REGION Network 20: Panel 20
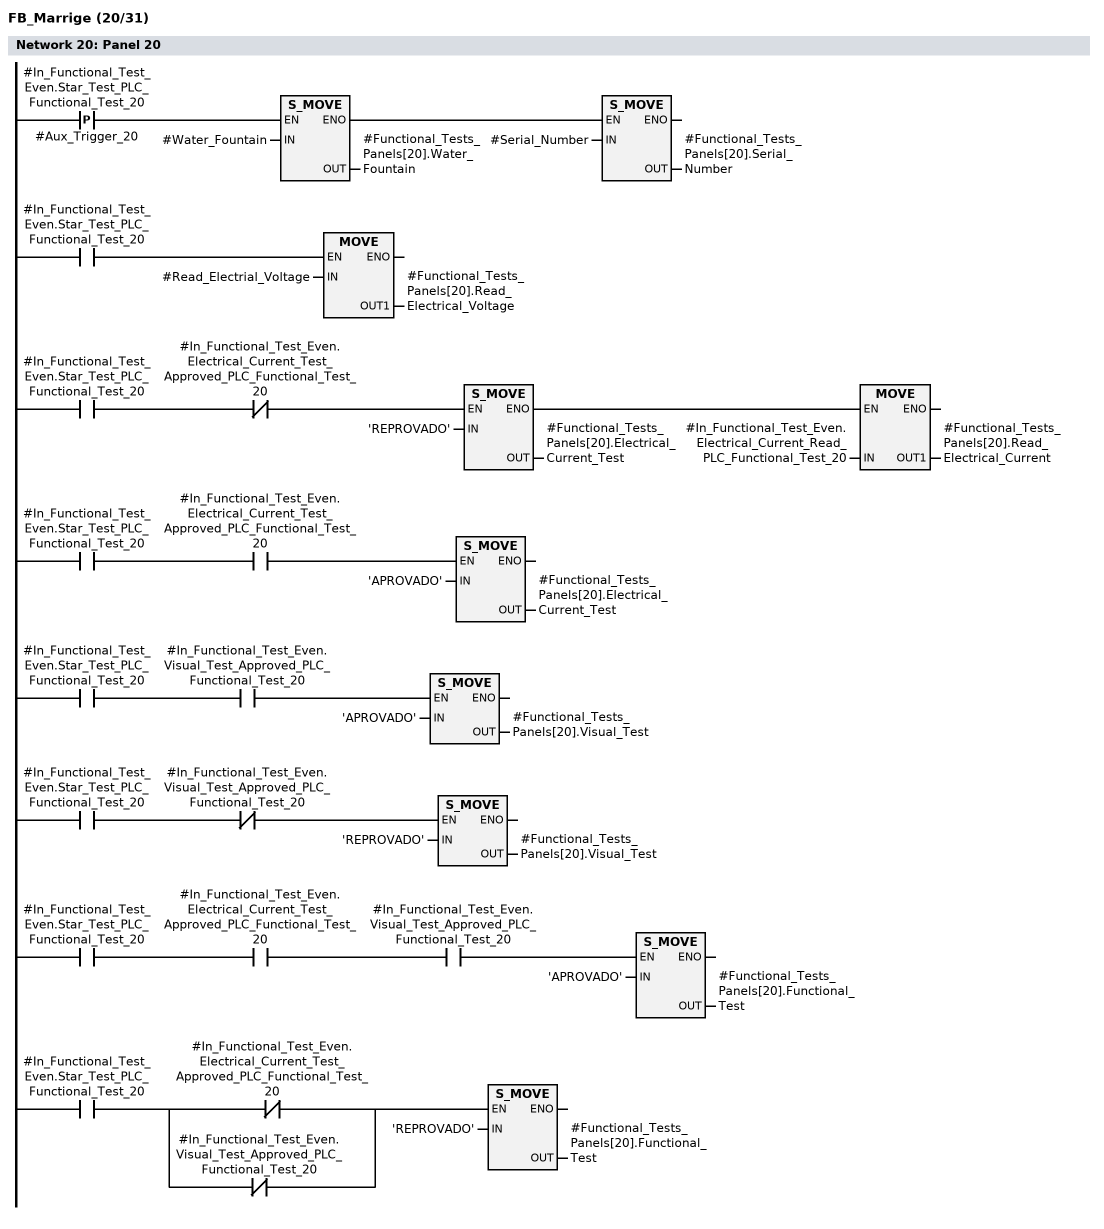
   RUNG wire#powerrail
      P_Contact(operand := #In_Functional_Test_Even.Star_Test_PLC_Functional_Test_20, bit := #Aux_Trigger_20)
      S_Move(in := #Water_Fountain, out => #Functional_Tests_Panels[20].Water_Fountain)
      S_Move(in := #Serial_Number, out => #Functional_Tests_Panels[20].Serial_Number)
   END_RUNG
   RUNG wire#powerrail
      Contact( #In_Functional_Test_Even.Star_Test_PLC_Functional_Test_20 )
      Move(in := #Read_Electrial_Voltage, out1 => #Functional_Tests_Panels[20].Read_Electrical_Voltage)
   END_RUNG
   RUNG wire#powerrail
      Contact( #In_Functional_Test_Even.Star_Test_PLC_Functional_Test_20 )
      I_Contact( #In_Functional_Test_Even.Electrical_Current_Test_Approved_PLC_Functional_Test_20 )
      S_Move(in := 'REPROVADO', out => #Functional_Tests_Panels[20].Electrical_Current_Test)
      Move(in := #In_Functional_Test_Even.Electrical_Current_Read_PLC_Functional_Test_20, out1 => #Functional_Tests_Panels[20].Read_Electrical_Current)
   END_RUNG
   RUNG wire#powerrail
      Contact( #In_Functional_Test_Even.Star_Test_PLC_Functional_Test_20 )
      Contact( #In_Functional_Test_Even.Electrical_Current_Test_Approved_PLC_Functional_Test_20 )
      S_Move(in := 'APROVADO', out => #Functional_Tests_Panels[20].Electrical_Current_Test)
   END_RUNG
   RUNG wire#powerrail
      Contact( #In_Functional_Test_Even.Star_Test_PLC_Functional_Test_20 )
      Contact( #In_Functional_Test_Even.Visual_Test_Approved_PLC_Functional_Test_20 )
      S_Move(in := 'APROVADO', out => #Functional_Tests_Panels[20].Visual_Test)
   END_RUNG
   RUNG wire#powerrail
      Contact( #In_Functional_Test_Even.Star_Test_PLC_Functional_Test_20 )
      I_Contact( #In_Functional_Test_Even.Visual_Test_Approved_PLC_Functional_Test_20 )
      S_Move(in := 'REPROVADO', out => #Functional_Tests_Panels[20].Visual_Test)
   END_RUNG
   RUNG wire#powerrail
      Contact( #In_Functional_Test_Even.Star_Test_PLC_Functional_Test_20 )
      Contact( #In_Functional_Test_Even.Electrical_Current_Test_Approved_PLC_Functional_Test_20 )
      Contact( #In_Functional_Test_Even.Visual_Test_Approved_PLC_Functional_Test_20 )
      S_Move(in := 'APROVADO', out => #Functional_Tests_Panels[20].Functional_Test)
   END_RUNG
   RUNG wire#powerrail
      Contact( #In_Functional_Test_Even.Star_Test_PLC_Functional_Test_20 )
      wire#w1
      I_Contact( #In_Functional_Test_Even.Electrical_Current_Test_Approved_PLC_Functional_Test_20 )
      wire#w2
      S_Move(in := 'REPROVADO', out => #Functional_Tests_Panels[20].Functional_Test)
   END_RUNG
   RUNG wire#w1
      I_Contact( #In_Functional_Test_Even.Visual_Test_Approved_PLC_Functional_Test_20 )
   END_RUNG wire#w2
   // the same network as SCL:
   #_w1 := #In_Functional_Test_Even.Star_Test_PLC_Functional_Test_20 AND NOT #Aux_Trigger_20;   // rising edge of #In_Functional_Test_Even.Star_Test_PLC_Functional_Test_20
   #Aux_Trigger_20 := #In_Functional_Test_Even.Star_Test_PLC_Functional_Test_20;
   IF #_w1 THEN
       #Functional_Tests_Panels[20].Water_Fountain := #Water_Fountain;
       #Functional_Tests_Panels[20].Serial_Number := #Serial_Number;
   END_IF;
   IF #In_Functional_Test_Even.Star_Test_PLC_Functional_Test_20 THEN
       #Functional_Tests_Panels[20].Read_Electrical_Voltage := #Read_Electrial_Voltage;
   END_IF;
   IF #In_Functional_Test_Even.Star_Test_PLC_Functional_Test_20 AND NOT #In_Functional_Test_Even.Electrical_Current_Test_Approved_PLC_Functional_Test_20 THEN
       #Functional_Tests_Panels[20].Electrical_Current_Test := 'REPROVADO';
       #Functional_Tests_Panels[20].Read_Electrical_Current := #In_Functional_Test_Even.Electrical_Current_Read_PLC_Functional_Test_20;
   END_IF;
   IF #In_Functional_Test_Even.Star_Test_PLC_Functional_Test_20 AND #In_Functional_Test_Even.Electrical_Current_Test_Approved_PLC_Functional_Test_20 THEN
       #Functional_Tests_Panels[20].Electrical_Current_Test := 'APROVADO';
   END_IF;
   IF #In_Functional_Test_Even.Star_Test_PLC_Functional_Test_20 AND #In_Functional_Test_Even.Visual_Test_Approved_PLC_Functional_Test_20 THEN
       #Functional_Tests_Panels[20].Visual_Test := 'APROVADO';
   END_IF;
   IF #In_Functional_Test_Even.Star_Test_PLC_Functional_Test_20 AND NOT #In_Functional_Test_Even.Visual_Test_Approved_PLC_Functional_Test_20 THEN
       #Functional_Tests_Panels[20].Visual_Test := 'REPROVADO';
   END_IF;
   IF #In_Functional_Test_Even.Star_Test_PLC_Functional_Test_20 AND #In_Functional_Test_Even.Electrical_Current_Test_Approved_PLC_Functional_Test_20 AND #In_Functional_Test_Even.Visual_Test_Approved_PLC_Functional_Test_20 THEN
       #Functional_Tests_Panels[20].Functional_Test := 'APROVADO';
   END_IF;
   IF #In_Functional_Test_Even.Star_Test_PLC_Functional_Test_20 AND (NOT #In_Functional_Test_Even.Electrical_Current_Test_Approved_PLC_Functional_Test_20 OR NOT #In_Functional_Test_Even.Visual_Test_Approved_PLC_Functional_Test_20) THEN
       #Functional_Tests_Panels[20].Functional_Test := 'REPROVADO';
   END_IF;
END_REGION

REGION Network 21: Panel 21
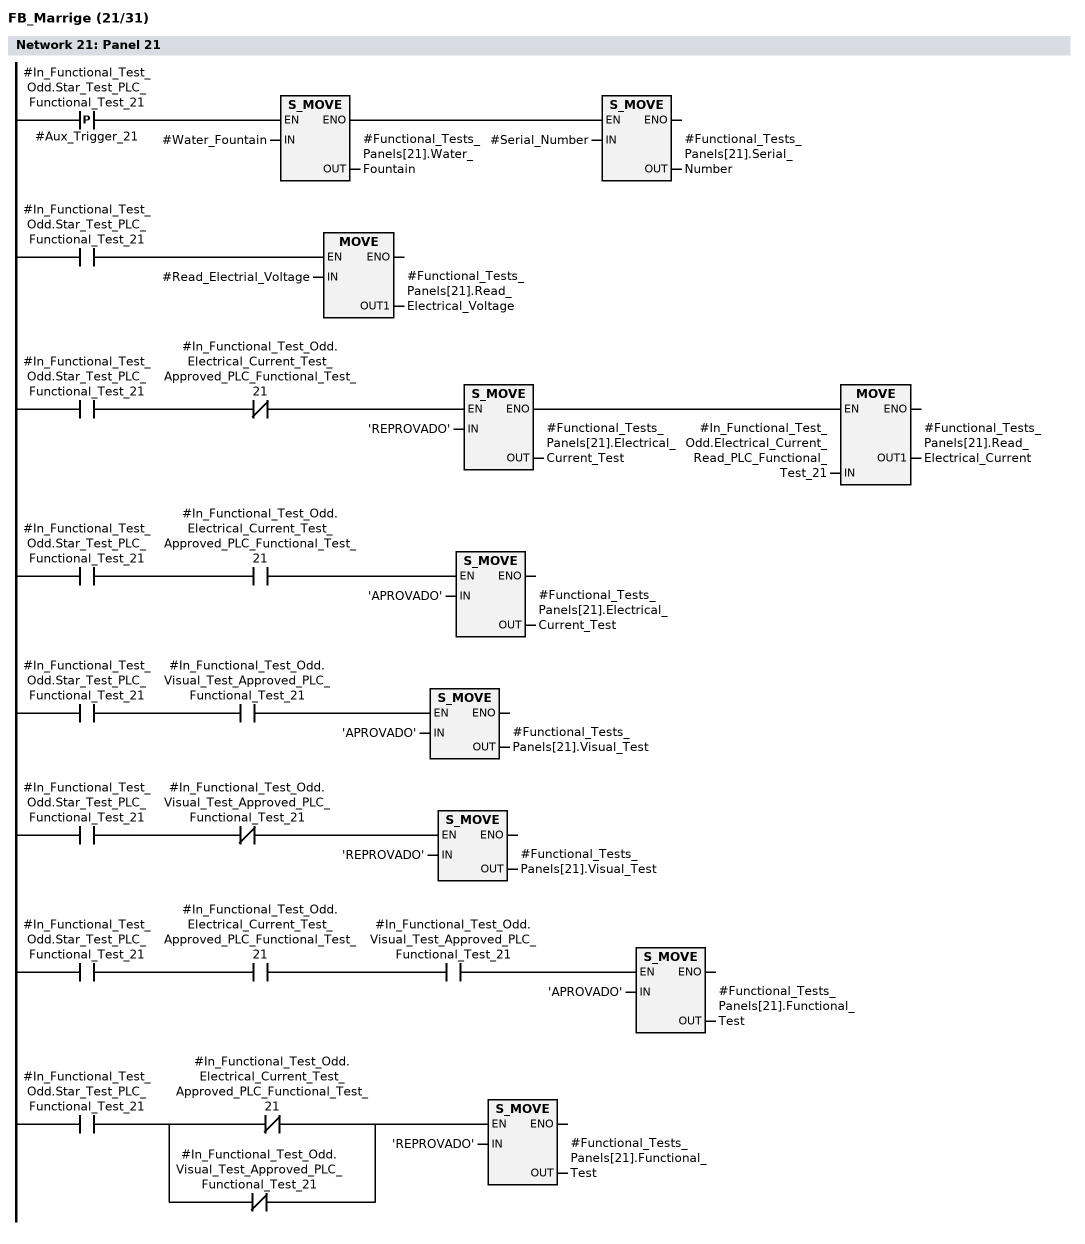
   RUNG wire#powerrail
      P_Contact(operand := #In_Functional_Test_Odd.Star_Test_PLC_Functional_Test_21, bit := #Aux_Trigger_21)
      S_Move(in := #Water_Fountain, out => #Functional_Tests_Panels[21].Water_Fountain)
      S_Move(in := #Serial_Number, out => #Functional_Tests_Panels[21].Serial_Number)
   END_RUNG
   RUNG wire#powerrail
      Contact( #In_Functional_Test_Odd.Star_Test_PLC_Functional_Test_21 )
      Move(in := #Read_Electrial_Voltage, out1 => #Functional_Tests_Panels[21].Read_Electrical_Voltage)
   END_RUNG
   RUNG wire#powerrail
      Contact( #In_Functional_Test_Odd.Star_Test_PLC_Functional_Test_21 )
      I_Contact( #In_Functional_Test_Odd.Electrical_Current_Test_Approved_PLC_Functional_Test_21 )
      S_Move(in := 'REPROVADO', out => #Functional_Tests_Panels[21].Electrical_Current_Test)
      Move(in := #In_Functional_Test_Odd.Electrical_Current_Read_PLC_Functional_Test_21, out1 => #Functional_Tests_Panels[21].Read_Electrical_Current)
   END_RUNG
   RUNG wire#powerrail
      Contact( #In_Functional_Test_Odd.Star_Test_PLC_Functional_Test_21 )
      Contact( #In_Functional_Test_Odd.Electrical_Current_Test_Approved_PLC_Functional_Test_21 )
      S_Move(in := 'APROVADO', out => #Functional_Tests_Panels[21].Electrical_Current_Test)
   END_RUNG
   RUNG wire#powerrail
      Contact( #In_Functional_Test_Odd.Star_Test_PLC_Functional_Test_21 )
      Contact( #In_Functional_Test_Odd.Visual_Test_Approved_PLC_Functional_Test_21 )
      S_Move(in := 'APROVADO', out => #Functional_Tests_Panels[21].Visual_Test)
   END_RUNG
   RUNG wire#powerrail
      Contact( #In_Functional_Test_Odd.Star_Test_PLC_Functional_Test_21 )
      I_Contact( #In_Functional_Test_Odd.Visual_Test_Approved_PLC_Functional_Test_21 )
      S_Move(in := 'REPROVADO', out => #Functional_Tests_Panels[21].Visual_Test)
   END_RUNG
   RUNG wire#powerrail
      Contact( #In_Functional_Test_Odd.Star_Test_PLC_Functional_Test_21 )
      Contact( #In_Functional_Test_Odd.Electrical_Current_Test_Approved_PLC_Functional_Test_21 )
      Contact( #In_Functional_Test_Odd.Visual_Test_Approved_PLC_Functional_Test_21 )
      S_Move(in := 'APROVADO', out => #Functional_Tests_Panels[21].Functional_Test)
   END_RUNG
   RUNG wire#powerrail
      Contact( #In_Functional_Test_Odd.Star_Test_PLC_Functional_Test_21 )
      wire#w1
      I_Contact( #In_Functional_Test_Odd.Electrical_Current_Test_Approved_PLC_Functional_Test_21 )
      wire#w2
      S_Move(in := 'REPROVADO', out => #Functional_Tests_Panels[21].Functional_Test)
   END_RUNG
   RUNG wire#w1
      I_Contact( #In_Functional_Test_Odd.Visual_Test_Approved_PLC_Functional_Test_21 )
   END_RUNG wire#w2
   // the same network as SCL:
   #_w1 := #In_Functional_Test_Odd.Star_Test_PLC_Functional_Test_21 AND NOT #Aux_Trigger_21;   // rising edge of #In_Functional_Test_Odd.Star_Test_PLC_Functional_Test_21
   #Aux_Trigger_21 := #In_Functional_Test_Odd.Star_Test_PLC_Functional_Test_21;
   IF #_w1 THEN
       #Functional_Tests_Panels[21].Water_Fountain := #Water_Fountain;
       #Functional_Tests_Panels[21].Serial_Number := #Serial_Number;
   END_IF;
   IF #In_Functional_Test_Odd.Star_Test_PLC_Functional_Test_21 THEN
       #Functional_Tests_Panels[21].Read_Electrical_Voltage := #Read_Electrial_Voltage;
   END_IF;
   IF #In_Functional_Test_Odd.Star_Test_PLC_Functional_Test_21 AND NOT #In_Functional_Test_Odd.Electrical_Current_Test_Approved_PLC_Functional_Test_21 THEN
       #Functional_Tests_Panels[21].Electrical_Current_Test := 'REPROVADO';
       #Functional_Tests_Panels[21].Read_Electrical_Current := #In_Functional_Test_Odd.Electrical_Current_Read_PLC_Functional_Test_21;
   END_IF;
   IF #In_Functional_Test_Odd.Star_Test_PLC_Functional_Test_21 AND #In_Functional_Test_Odd.Electrical_Current_Test_Approved_PLC_Functional_Test_21 THEN
       #Functional_Tests_Panels[21].Electrical_Current_Test := 'APROVADO';
   END_IF;
   IF #In_Functional_Test_Odd.Star_Test_PLC_Functional_Test_21 AND #In_Functional_Test_Odd.Visual_Test_Approved_PLC_Functional_Test_21 THEN
       #Functional_Tests_Panels[21].Visual_Test := 'APROVADO';
   END_IF;
   IF #In_Functional_Test_Odd.Star_Test_PLC_Functional_Test_21 AND NOT #In_Functional_Test_Odd.Visual_Test_Approved_PLC_Functional_Test_21 THEN
       #Functional_Tests_Panels[21].Visual_Test := 'REPROVADO';
   END_IF;
   IF #In_Functional_Test_Odd.Star_Test_PLC_Functional_Test_21 AND #In_Functional_Test_Odd.Electrical_Current_Test_Approved_PLC_Functional_Test_21 AND #In_Functional_Test_Odd.Visual_Test_Approved_PLC_Functional_Test_21 THEN
       #Functional_Tests_Panels[21].Functional_Test := 'APROVADO';
   END_IF;
   IF #In_Functional_Test_Odd.Star_Test_PLC_Functional_Test_21 AND (NOT #In_Functional_Test_Odd.Electrical_Current_Test_Approved_PLC_Functional_Test_21 OR NOT #In_Functional_Test_Odd.Visual_Test_Approved_PLC_Functional_Test_21) THEN
       #Functional_Tests_Panels[21].Functional_Test := 'REPROVADO';
   END_IF;
END_REGION

REGION Network 22: Panel 22
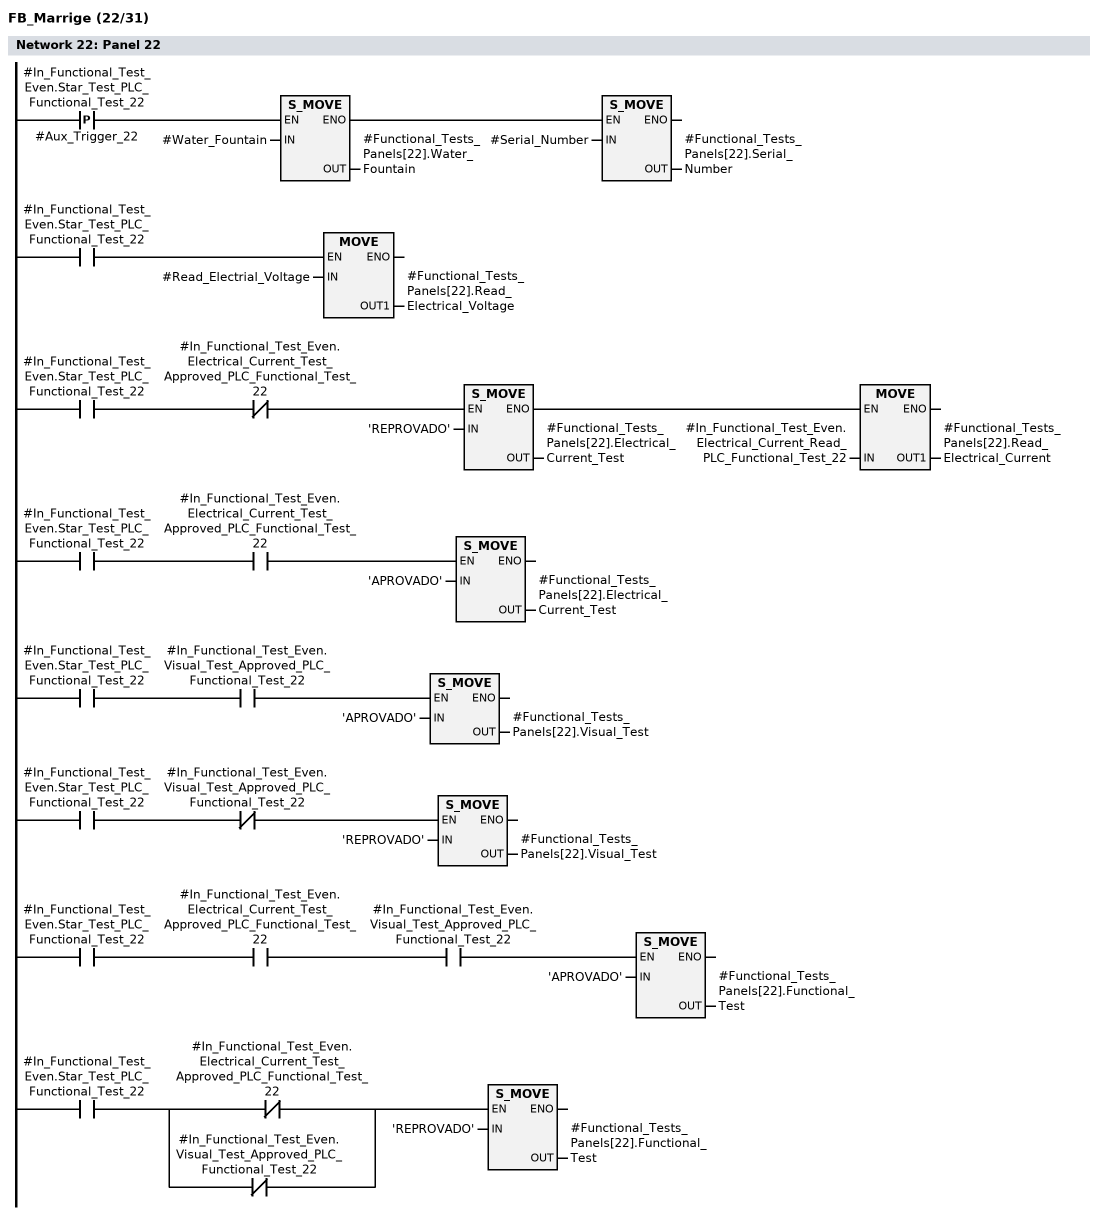
   RUNG wire#powerrail
      P_Contact(operand := #In_Functional_Test_Even.Star_Test_PLC_Functional_Test_22, bit := #Aux_Trigger_22)
      S_Move(in := #Water_Fountain, out => #Functional_Tests_Panels[22].Water_Fountain)
      S_Move(in := #Serial_Number, out => #Functional_Tests_Panels[22].Serial_Number)
   END_RUNG
   RUNG wire#powerrail
      Contact( #In_Functional_Test_Even.Star_Test_PLC_Functional_Test_22 )
      Move(in := #Read_Electrial_Voltage, out1 => #Functional_Tests_Panels[22].Read_Electrical_Voltage)
   END_RUNG
   RUNG wire#powerrail
      Contact( #In_Functional_Test_Even.Star_Test_PLC_Functional_Test_22 )
      I_Contact( #In_Functional_Test_Even.Electrical_Current_Test_Approved_PLC_Functional_Test_22 )
      S_Move(in := 'REPROVADO', out => #Functional_Tests_Panels[22].Electrical_Current_Test)
      Move(in := #In_Functional_Test_Even.Electrical_Current_Read_PLC_Functional_Test_22, out1 => #Functional_Tests_Panels[22].Read_Electrical_Current)
   END_RUNG
   RUNG wire#powerrail
      Contact( #In_Functional_Test_Even.Star_Test_PLC_Functional_Test_22 )
      Contact( #In_Functional_Test_Even.Electrical_Current_Test_Approved_PLC_Functional_Test_22 )
      S_Move(in := 'APROVADO', out => #Functional_Tests_Panels[22].Electrical_Current_Test)
   END_RUNG
   RUNG wire#powerrail
      Contact( #In_Functional_Test_Even.Star_Test_PLC_Functional_Test_22 )
      Contact( #In_Functional_Test_Even.Visual_Test_Approved_PLC_Functional_Test_22 )
      S_Move(in := 'APROVADO', out => #Functional_Tests_Panels[22].Visual_Test)
   END_RUNG
   RUNG wire#powerrail
      Contact( #In_Functional_Test_Even.Star_Test_PLC_Functional_Test_22 )
      I_Contact( #In_Functional_Test_Even.Visual_Test_Approved_PLC_Functional_Test_22 )
      S_Move(in := 'REPROVADO', out => #Functional_Tests_Panels[22].Visual_Test)
   END_RUNG
   RUNG wire#powerrail
      Contact( #In_Functional_Test_Even.Star_Test_PLC_Functional_Test_22 )
      Contact( #In_Functional_Test_Even.Electrical_Current_Test_Approved_PLC_Functional_Test_22 )
      Contact( #In_Functional_Test_Even.Visual_Test_Approved_PLC_Functional_Test_22 )
      S_Move(in := 'APROVADO', out => #Functional_Tests_Panels[22].Functional_Test)
   END_RUNG
   RUNG wire#powerrail
      Contact( #In_Functional_Test_Even.Star_Test_PLC_Functional_Test_22 )
      wire#w1
      I_Contact( #In_Functional_Test_Even.Electrical_Current_Test_Approved_PLC_Functional_Test_22 )
      wire#w2
      S_Move(in := 'REPROVADO', out => #Functional_Tests_Panels[22].Functional_Test)
   END_RUNG
   RUNG wire#w1
      I_Contact( #In_Functional_Test_Even.Visual_Test_Approved_PLC_Functional_Test_22 )
   END_RUNG wire#w2
   // the same network as SCL:
   #_w1 := #In_Functional_Test_Even.Star_Test_PLC_Functional_Test_22 AND NOT #Aux_Trigger_22;   // rising edge of #In_Functional_Test_Even.Star_Test_PLC_Functional_Test_22
   #Aux_Trigger_22 := #In_Functional_Test_Even.Star_Test_PLC_Functional_Test_22;
   IF #_w1 THEN
       #Functional_Tests_Panels[22].Water_Fountain := #Water_Fountain;
       #Functional_Tests_Panels[22].Serial_Number := #Serial_Number;
   END_IF;
   IF #In_Functional_Test_Even.Star_Test_PLC_Functional_Test_22 THEN
       #Functional_Tests_Panels[22].Read_Electrical_Voltage := #Read_Electrial_Voltage;
   END_IF;
   IF #In_Functional_Test_Even.Star_Test_PLC_Functional_Test_22 AND NOT #In_Functional_Test_Even.Electrical_Current_Test_Approved_PLC_Functional_Test_22 THEN
       #Functional_Tests_Panels[22].Electrical_Current_Test := 'REPROVADO';
       #Functional_Tests_Panels[22].Read_Electrical_Current := #In_Functional_Test_Even.Electrical_Current_Read_PLC_Functional_Test_22;
   END_IF;
   IF #In_Functional_Test_Even.Star_Test_PLC_Functional_Test_22 AND #In_Functional_Test_Even.Electrical_Current_Test_Approved_PLC_Functional_Test_22 THEN
       #Functional_Tests_Panels[22].Electrical_Current_Test := 'APROVADO';
   END_IF;
   IF #In_Functional_Test_Even.Star_Test_PLC_Functional_Test_22 AND #In_Functional_Test_Even.Visual_Test_Approved_PLC_Functional_Test_22 THEN
       #Functional_Tests_Panels[22].Visual_Test := 'APROVADO';
   END_IF;
   IF #In_Functional_Test_Even.Star_Test_PLC_Functional_Test_22 AND NOT #In_Functional_Test_Even.Visual_Test_Approved_PLC_Functional_Test_22 THEN
       #Functional_Tests_Panels[22].Visual_Test := 'REPROVADO';
   END_IF;
   IF #In_Functional_Test_Even.Star_Test_PLC_Functional_Test_22 AND #In_Functional_Test_Even.Electrical_Current_Test_Approved_PLC_Functional_Test_22 AND #In_Functional_Test_Even.Visual_Test_Approved_PLC_Functional_Test_22 THEN
       #Functional_Tests_Panels[22].Functional_Test := 'APROVADO';
   END_IF;
   IF #In_Functional_Test_Even.Star_Test_PLC_Functional_Test_22 AND (NOT #In_Functional_Test_Even.Electrical_Current_Test_Approved_PLC_Functional_Test_22 OR NOT #In_Functional_Test_Even.Visual_Test_Approved_PLC_Functional_Test_22) THEN
       #Functional_Tests_Panels[22].Functional_Test := 'REPROVADO';
   END_IF;
END_REGION

REGION Network 23: Panel 23
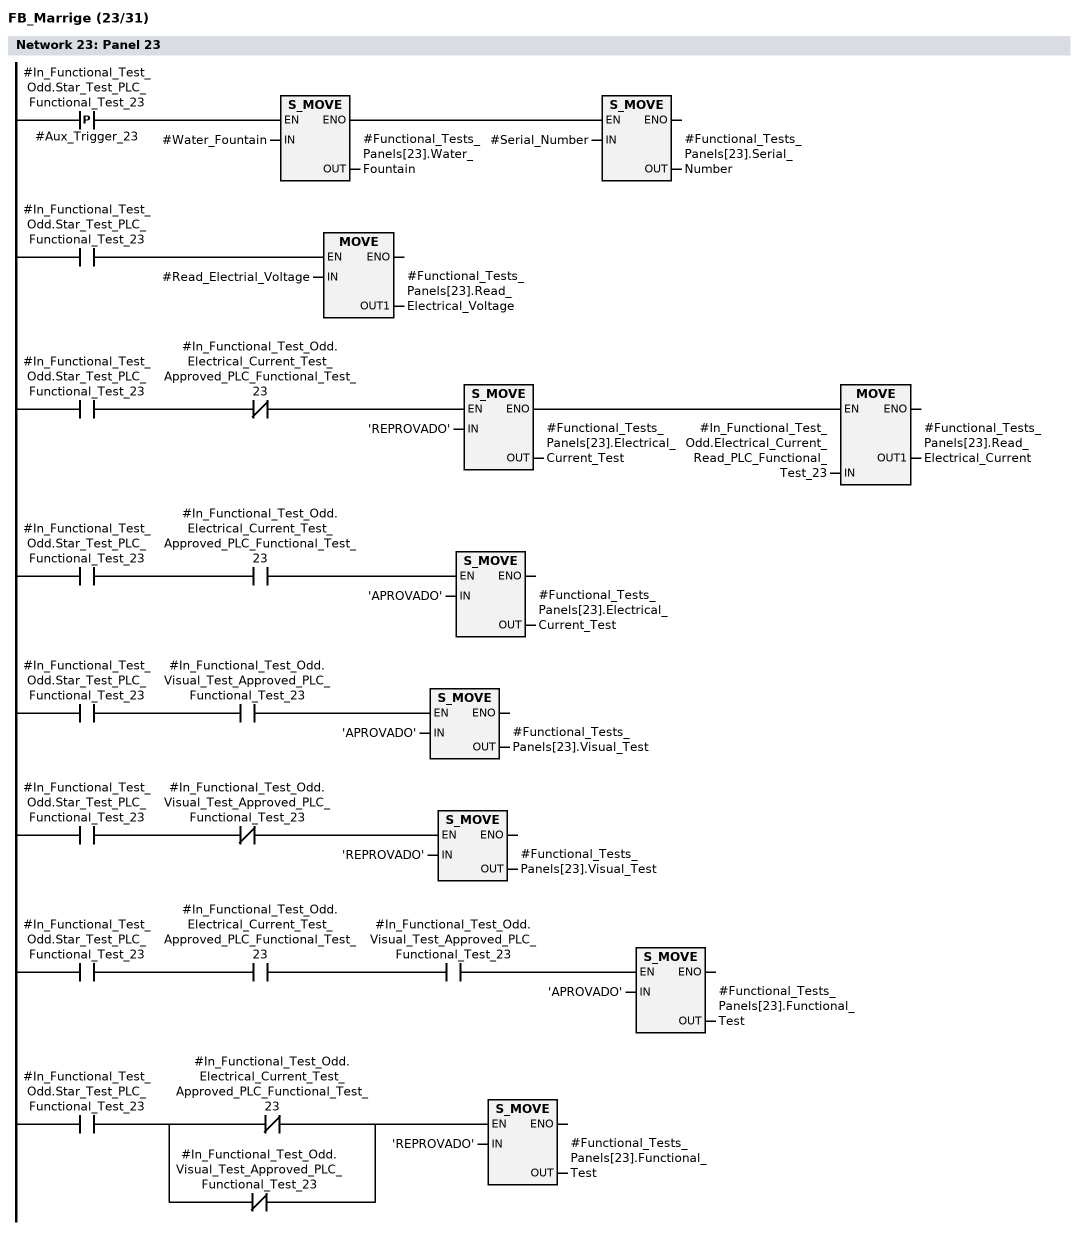
   RUNG wire#powerrail
      P_Contact(operand := #In_Functional_Test_Odd.Star_Test_PLC_Functional_Test_23, bit := #Aux_Trigger_23)
      S_Move(in := #Water_Fountain, out => #Functional_Tests_Panels[23].Water_Fountain)
      S_Move(in := #Serial_Number, out => #Functional_Tests_Panels[23].Serial_Number)
   END_RUNG
   RUNG wire#powerrail
      Contact( #In_Functional_Test_Odd.Star_Test_PLC_Functional_Test_23 )
      Move(in := #Read_Electrial_Voltage, out1 => #Functional_Tests_Panels[23].Read_Electrical_Voltage)
   END_RUNG
   RUNG wire#powerrail
      Contact( #In_Functional_Test_Odd.Star_Test_PLC_Functional_Test_23 )
      I_Contact( #In_Functional_Test_Odd.Electrical_Current_Test_Approved_PLC_Functional_Test_23 )
      S_Move(in := 'REPROVADO', out => #Functional_Tests_Panels[23].Electrical_Current_Test)
      Move(in := #In_Functional_Test_Odd.Electrical_Current_Read_PLC_Functional_Test_23, out1 => #Functional_Tests_Panels[23].Read_Electrical_Current)
   END_RUNG
   RUNG wire#powerrail
      Contact( #In_Functional_Test_Odd.Star_Test_PLC_Functional_Test_23 )
      Contact( #In_Functional_Test_Odd.Electrical_Current_Test_Approved_PLC_Functional_Test_23 )
      S_Move(in := 'APROVADO', out => #Functional_Tests_Panels[23].Electrical_Current_Test)
   END_RUNG
   RUNG wire#powerrail
      Contact( #In_Functional_Test_Odd.Star_Test_PLC_Functional_Test_23 )
      Contact( #In_Functional_Test_Odd.Visual_Test_Approved_PLC_Functional_Test_23 )
      S_Move(in := 'APROVADO', out => #Functional_Tests_Panels[23].Visual_Test)
   END_RUNG
   RUNG wire#powerrail
      Contact( #In_Functional_Test_Odd.Star_Test_PLC_Functional_Test_23 )
      I_Contact( #In_Functional_Test_Odd.Visual_Test_Approved_PLC_Functional_Test_23 )
      S_Move(in := 'REPROVADO', out => #Functional_Tests_Panels[23].Visual_Test)
   END_RUNG
   RUNG wire#powerrail
      Contact( #In_Functional_Test_Odd.Star_Test_PLC_Functional_Test_23 )
      Contact( #In_Functional_Test_Odd.Electrical_Current_Test_Approved_PLC_Functional_Test_23 )
      Contact( #In_Functional_Test_Odd.Visual_Test_Approved_PLC_Functional_Test_23 )
      S_Move(in := 'APROVADO', out => #Functional_Tests_Panels[23].Functional_Test)
   END_RUNG
   RUNG wire#powerrail
      Contact( #In_Functional_Test_Odd.Star_Test_PLC_Functional_Test_23 )
      wire#w1
      I_Contact( #In_Functional_Test_Odd.Electrical_Current_Test_Approved_PLC_Functional_Test_23 )
      wire#w2
      S_Move(in := 'REPROVADO', out => #Functional_Tests_Panels[23].Functional_Test)
   END_RUNG
   RUNG wire#w1
      I_Contact( #In_Functional_Test_Odd.Visual_Test_Approved_PLC_Functional_Test_23 )
   END_RUNG wire#w2
   // the same network as SCL:
   #_w1 := #In_Functional_Test_Odd.Star_Test_PLC_Functional_Test_23 AND NOT #Aux_Trigger_23;   // rising edge of #In_Functional_Test_Odd.Star_Test_PLC_Functional_Test_23
   #Aux_Trigger_23 := #In_Functional_Test_Odd.Star_Test_PLC_Functional_Test_23;
   IF #_w1 THEN
       #Functional_Tests_Panels[23].Water_Fountain := #Water_Fountain;
       #Functional_Tests_Panels[23].Serial_Number := #Serial_Number;
   END_IF;
   IF #In_Functional_Test_Odd.Star_Test_PLC_Functional_Test_23 THEN
       #Functional_Tests_Panels[23].Read_Electrical_Voltage := #Read_Electrial_Voltage;
   END_IF;
   IF #In_Functional_Test_Odd.Star_Test_PLC_Functional_Test_23 AND NOT #In_Functional_Test_Odd.Electrical_Current_Test_Approved_PLC_Functional_Test_23 THEN
       #Functional_Tests_Panels[23].Electrical_Current_Test := 'REPROVADO';
       #Functional_Tests_Panels[23].Read_Electrical_Current := #In_Functional_Test_Odd.Electrical_Current_Read_PLC_Functional_Test_23;
   END_IF;
   IF #In_Functional_Test_Odd.Star_Test_PLC_Functional_Test_23 AND #In_Functional_Test_Odd.Electrical_Current_Test_Approved_PLC_Functional_Test_23 THEN
       #Functional_Tests_Panels[23].Electrical_Current_Test := 'APROVADO';
   END_IF;
   IF #In_Functional_Test_Odd.Star_Test_PLC_Functional_Test_23 AND #In_Functional_Test_Odd.Visual_Test_Approved_PLC_Functional_Test_23 THEN
       #Functional_Tests_Panels[23].Visual_Test := 'APROVADO';
   END_IF;
   IF #In_Functional_Test_Odd.Star_Test_PLC_Functional_Test_23 AND NOT #In_Functional_Test_Odd.Visual_Test_Approved_PLC_Functional_Test_23 THEN
       #Functional_Tests_Panels[23].Visual_Test := 'REPROVADO';
   END_IF;
   IF #In_Functional_Test_Odd.Star_Test_PLC_Functional_Test_23 AND #In_Functional_Test_Odd.Electrical_Current_Test_Approved_PLC_Functional_Test_23 AND #In_Functional_Test_Odd.Visual_Test_Approved_PLC_Functional_Test_23 THEN
       #Functional_Tests_Panels[23].Functional_Test := 'APROVADO';
   END_IF;
   IF #In_Functional_Test_Odd.Star_Test_PLC_Functional_Test_23 AND (NOT #In_Functional_Test_Odd.Electrical_Current_Test_Approved_PLC_Functional_Test_23 OR NOT #In_Functional_Test_Odd.Visual_Test_Approved_PLC_Functional_Test_23) THEN
       #Functional_Tests_Panels[23].Functional_Test := 'REPROVADO';
   END_IF;
END_REGION

REGION Network 24: Panel 24
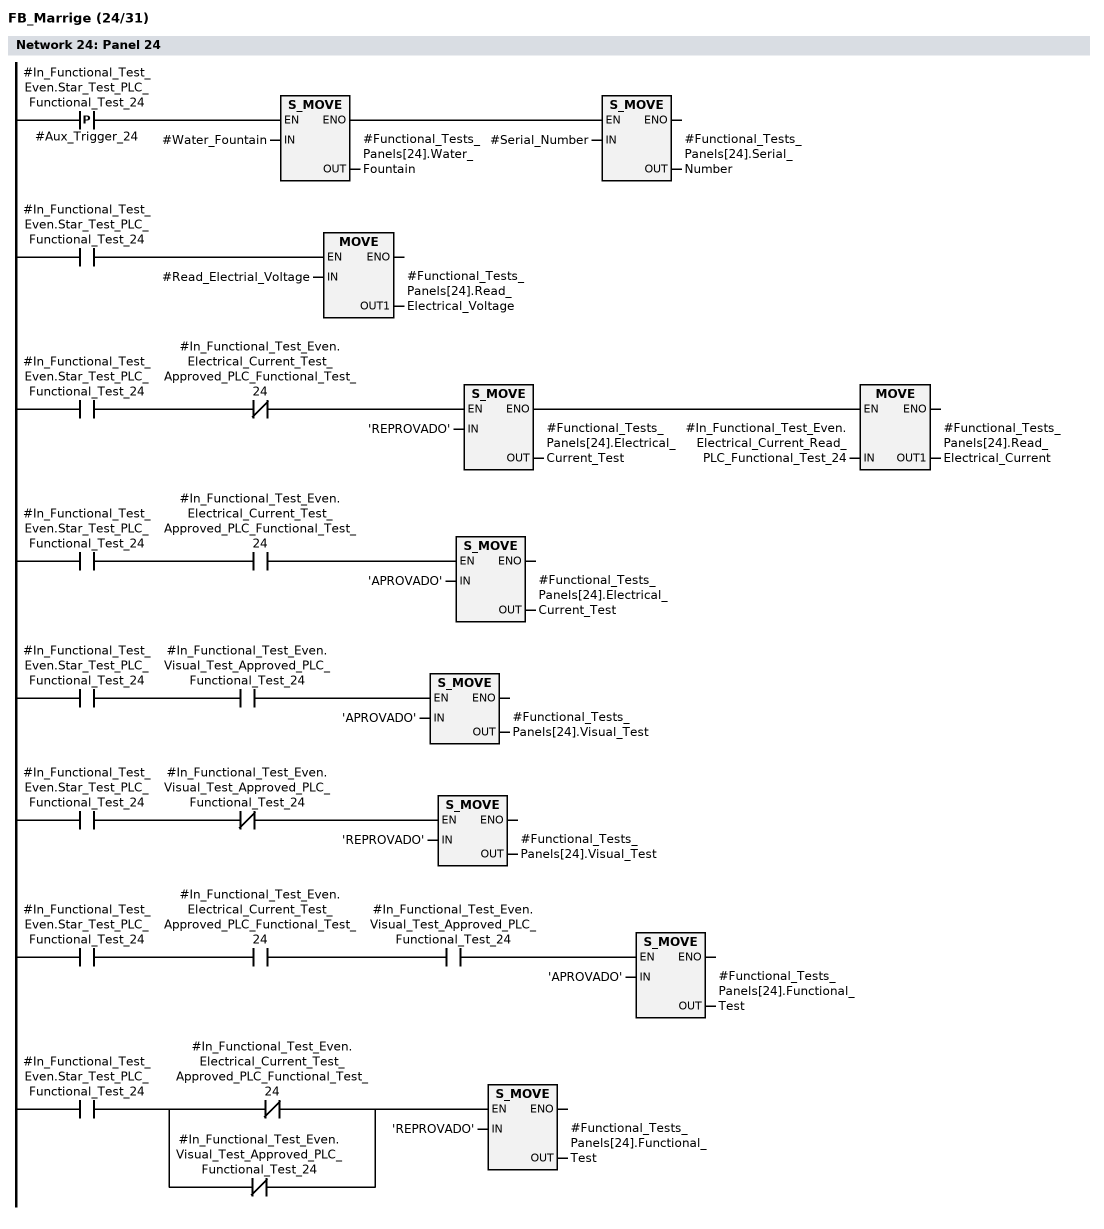
   RUNG wire#powerrail
      P_Contact(operand := #In_Functional_Test_Even.Star_Test_PLC_Functional_Test_24, bit := #Aux_Trigger_24)
      S_Move(in := #Water_Fountain, out => #Functional_Tests_Panels[24].Water_Fountain)
      S_Move(in := #Serial_Number, out => #Functional_Tests_Panels[24].Serial_Number)
   END_RUNG
   RUNG wire#powerrail
      Contact( #In_Functional_Test_Even.Star_Test_PLC_Functional_Test_24 )
      Move(in := #Read_Electrial_Voltage, out1 => #Functional_Tests_Panels[24].Read_Electrical_Voltage)
   END_RUNG
   RUNG wire#powerrail
      Contact( #In_Functional_Test_Even.Star_Test_PLC_Functional_Test_24 )
      I_Contact( #In_Functional_Test_Even.Electrical_Current_Test_Approved_PLC_Functional_Test_24 )
      S_Move(in := 'REPROVADO', out => #Functional_Tests_Panels[24].Electrical_Current_Test)
      Move(in := #In_Functional_Test_Even.Electrical_Current_Read_PLC_Functional_Test_24, out1 => #Functional_Tests_Panels[24].Read_Electrical_Current)
   END_RUNG
   RUNG wire#powerrail
      Contact( #In_Functional_Test_Even.Star_Test_PLC_Functional_Test_24 )
      Contact( #In_Functional_Test_Even.Electrical_Current_Test_Approved_PLC_Functional_Test_24 )
      S_Move(in := 'APROVADO', out => #Functional_Tests_Panels[24].Electrical_Current_Test)
   END_RUNG
   RUNG wire#powerrail
      Contact( #In_Functional_Test_Even.Star_Test_PLC_Functional_Test_24 )
      Contact( #In_Functional_Test_Even.Visual_Test_Approved_PLC_Functional_Test_24 )
      S_Move(in := 'APROVADO', out => #Functional_Tests_Panels[24].Visual_Test)
   END_RUNG
   RUNG wire#powerrail
      Contact( #In_Functional_Test_Even.Star_Test_PLC_Functional_Test_24 )
      I_Contact( #In_Functional_Test_Even.Visual_Test_Approved_PLC_Functional_Test_24 )
      S_Move(in := 'REPROVADO', out => #Functional_Tests_Panels[24].Visual_Test)
   END_RUNG
   RUNG wire#powerrail
      Contact( #In_Functional_Test_Even.Star_Test_PLC_Functional_Test_24 )
      Contact( #In_Functional_Test_Even.Electrical_Current_Test_Approved_PLC_Functional_Test_24 )
      Contact( #In_Functional_Test_Even.Visual_Test_Approved_PLC_Functional_Test_24 )
      S_Move(in := 'APROVADO', out => #Functional_Tests_Panels[24].Functional_Test)
   END_RUNG
   RUNG wire#powerrail
      Contact( #In_Functional_Test_Even.Star_Test_PLC_Functional_Test_24 )
      wire#w1
      I_Contact( #In_Functional_Test_Even.Electrical_Current_Test_Approved_PLC_Functional_Test_24 )
      wire#w2
      S_Move(in := 'REPROVADO', out => #Functional_Tests_Panels[24].Functional_Test)
   END_RUNG
   RUNG wire#w1
      I_Contact( #In_Functional_Test_Even.Visual_Test_Approved_PLC_Functional_Test_24 )
   END_RUNG wire#w2
   // the same network as SCL:
   #_w1 := #In_Functional_Test_Even.Star_Test_PLC_Functional_Test_24 AND NOT #Aux_Trigger_24;   // rising edge of #In_Functional_Test_Even.Star_Test_PLC_Functional_Test_24
   #Aux_Trigger_24 := #In_Functional_Test_Even.Star_Test_PLC_Functional_Test_24;
   IF #_w1 THEN
       #Functional_Tests_Panels[24].Water_Fountain := #Water_Fountain;
       #Functional_Tests_Panels[24].Serial_Number := #Serial_Number;
   END_IF;
   IF #In_Functional_Test_Even.Star_Test_PLC_Functional_Test_24 THEN
       #Functional_Tests_Panels[24].Read_Electrical_Voltage := #Read_Electrial_Voltage;
   END_IF;
   IF #In_Functional_Test_Even.Star_Test_PLC_Functional_Test_24 AND NOT #In_Functional_Test_Even.Electrical_Current_Test_Approved_PLC_Functional_Test_24 THEN
       #Functional_Tests_Panels[24].Electrical_Current_Test := 'REPROVADO';
       #Functional_Tests_Panels[24].Read_Electrical_Current := #In_Functional_Test_Even.Electrical_Current_Read_PLC_Functional_Test_24;
   END_IF;
   IF #In_Functional_Test_Even.Star_Test_PLC_Functional_Test_24 AND #In_Functional_Test_Even.Electrical_Current_Test_Approved_PLC_Functional_Test_24 THEN
       #Functional_Tests_Panels[24].Electrical_Current_Test := 'APROVADO';
   END_IF;
   IF #In_Functional_Test_Even.Star_Test_PLC_Functional_Test_24 AND #In_Functional_Test_Even.Visual_Test_Approved_PLC_Functional_Test_24 THEN
       #Functional_Tests_Panels[24].Visual_Test := 'APROVADO';
   END_IF;
   IF #In_Functional_Test_Even.Star_Test_PLC_Functional_Test_24 AND NOT #In_Functional_Test_Even.Visual_Test_Approved_PLC_Functional_Test_24 THEN
       #Functional_Tests_Panels[24].Visual_Test := 'REPROVADO';
   END_IF;
   IF #In_Functional_Test_Even.Star_Test_PLC_Functional_Test_24 AND #In_Functional_Test_Even.Electrical_Current_Test_Approved_PLC_Functional_Test_24 AND #In_Functional_Test_Even.Visual_Test_Approved_PLC_Functional_Test_24 THEN
       #Functional_Tests_Panels[24].Functional_Test := 'APROVADO';
   END_IF;
   IF #In_Functional_Test_Even.Star_Test_PLC_Functional_Test_24 AND (NOT #In_Functional_Test_Even.Electrical_Current_Test_Approved_PLC_Functional_Test_24 OR NOT #In_Functional_Test_Even.Visual_Test_Approved_PLC_Functional_Test_24) THEN
       #Functional_Tests_Panels[24].Functional_Test := 'REPROVADO';
   END_IF;
END_REGION

REGION Network 25: Panel 25
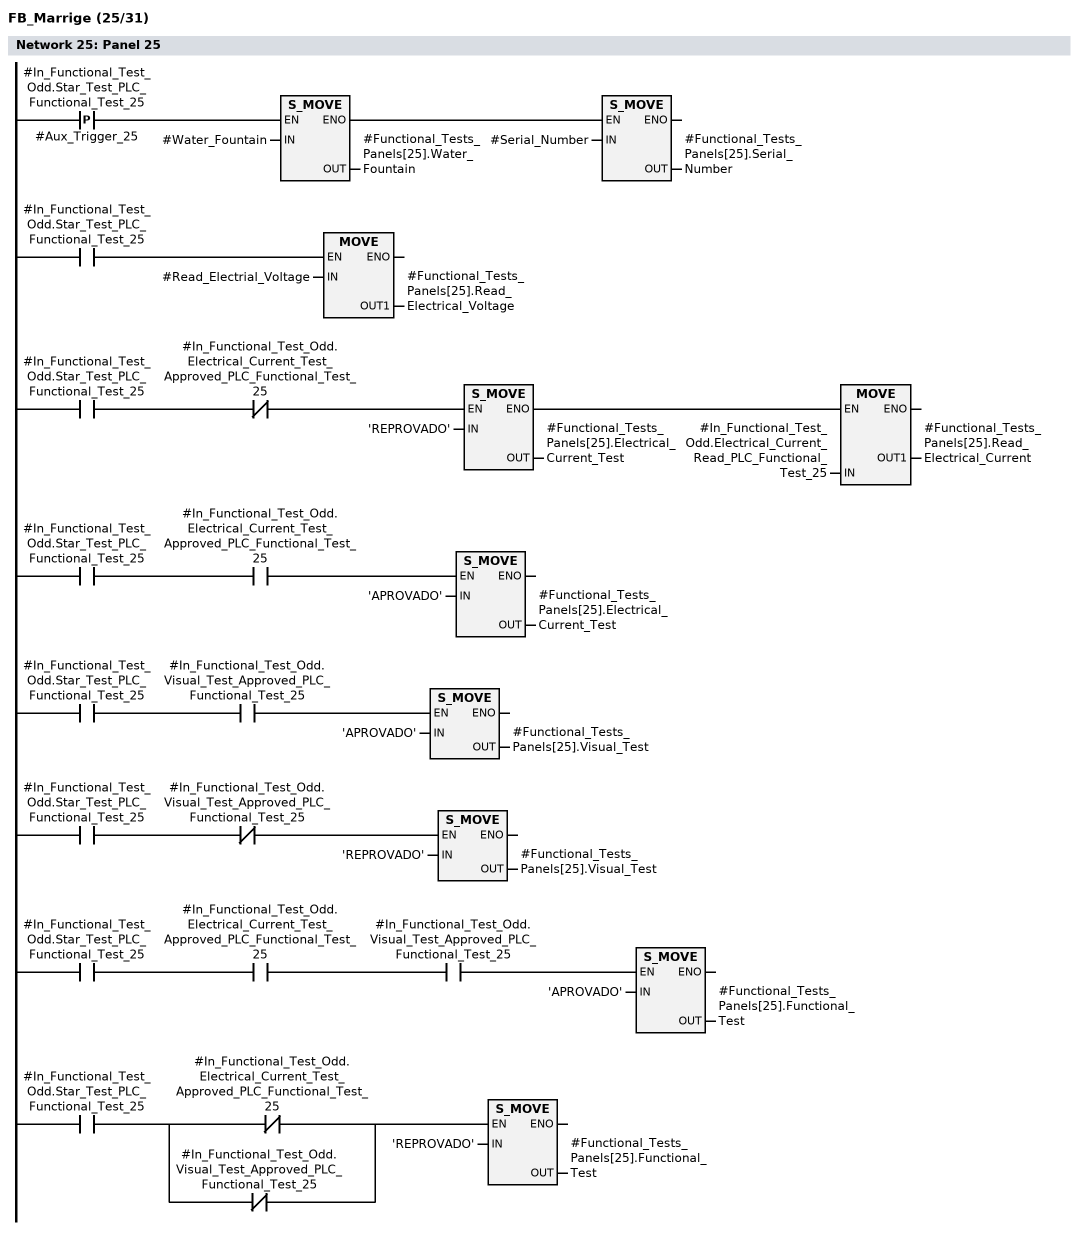
   RUNG wire#powerrail
      P_Contact(operand := #In_Functional_Test_Odd.Star_Test_PLC_Functional_Test_25, bit := #Aux_Trigger_25)
      S_Move(in := #Water_Fountain, out => #Functional_Tests_Panels[25].Water_Fountain)
      S_Move(in := #Serial_Number, out => #Functional_Tests_Panels[25].Serial_Number)
   END_RUNG
   RUNG wire#powerrail
      Contact( #In_Functional_Test_Odd.Star_Test_PLC_Functional_Test_25 )
      Move(in := #Read_Electrial_Voltage, out1 => #Functional_Tests_Panels[25].Read_Electrical_Voltage)
   END_RUNG
   RUNG wire#powerrail
      Contact( #In_Functional_Test_Odd.Star_Test_PLC_Functional_Test_25 )
      I_Contact( #In_Functional_Test_Odd.Electrical_Current_Test_Approved_PLC_Functional_Test_25 )
      S_Move(in := 'REPROVADO', out => #Functional_Tests_Panels[25].Electrical_Current_Test)
      Move(in := #In_Functional_Test_Odd.Electrical_Current_Read_PLC_Functional_Test_25, out1 => #Functional_Tests_Panels[25].Read_Electrical_Current)
   END_RUNG
   RUNG wire#powerrail
      Contact( #In_Functional_Test_Odd.Star_Test_PLC_Functional_Test_25 )
      Contact( #In_Functional_Test_Odd.Electrical_Current_Test_Approved_PLC_Functional_Test_25 )
      S_Move(in := 'APROVADO', out => #Functional_Tests_Panels[25].Electrical_Current_Test)
   END_RUNG
   RUNG wire#powerrail
      Contact( #In_Functional_Test_Odd.Star_Test_PLC_Functional_Test_25 )
      Contact( #In_Functional_Test_Odd.Visual_Test_Approved_PLC_Functional_Test_25 )
      S_Move(in := 'APROVADO', out => #Functional_Tests_Panels[25].Visual_Test)
   END_RUNG
   RUNG wire#powerrail
      Contact( #In_Functional_Test_Odd.Star_Test_PLC_Functional_Test_25 )
      I_Contact( #In_Functional_Test_Odd.Visual_Test_Approved_PLC_Functional_Test_25 )
      S_Move(in := 'REPROVADO', out => #Functional_Tests_Panels[25].Visual_Test)
   END_RUNG
   RUNG wire#powerrail
      Contact( #In_Functional_Test_Odd.Star_Test_PLC_Functional_Test_25 )
      Contact( #In_Functional_Test_Odd.Electrical_Current_Test_Approved_PLC_Functional_Test_25 )
      Contact( #In_Functional_Test_Odd.Visual_Test_Approved_PLC_Functional_Test_25 )
      S_Move(in := 'APROVADO', out => #Functional_Tests_Panels[25].Functional_Test)
   END_RUNG
   RUNG wire#powerrail
      Contact( #In_Functional_Test_Odd.Star_Test_PLC_Functional_Test_25 )
      wire#w1
      I_Contact( #In_Functional_Test_Odd.Electrical_Current_Test_Approved_PLC_Functional_Test_25 )
      wire#w2
      S_Move(in := 'REPROVADO', out => #Functional_Tests_Panels[25].Functional_Test)
   END_RUNG
   RUNG wire#w1
      I_Contact( #In_Functional_Test_Odd.Visual_Test_Approved_PLC_Functional_Test_25 )
   END_RUNG wire#w2
   // the same network as SCL:
   #_w1 := #In_Functional_Test_Odd.Star_Test_PLC_Functional_Test_25 AND NOT #Aux_Trigger_25;   // rising edge of #In_Functional_Test_Odd.Star_Test_PLC_Functional_Test_25
   #Aux_Trigger_25 := #In_Functional_Test_Odd.Star_Test_PLC_Functional_Test_25;
   IF #_w1 THEN
       #Functional_Tests_Panels[25].Water_Fountain := #Water_Fountain;
       #Functional_Tests_Panels[25].Serial_Number := #Serial_Number;
   END_IF;
   IF #In_Functional_Test_Odd.Star_Test_PLC_Functional_Test_25 THEN
       #Functional_Tests_Panels[25].Read_Electrical_Voltage := #Read_Electrial_Voltage;
   END_IF;
   IF #In_Functional_Test_Odd.Star_Test_PLC_Functional_Test_25 AND NOT #In_Functional_Test_Odd.Electrical_Current_Test_Approved_PLC_Functional_Test_25 THEN
       #Functional_Tests_Panels[25].Electrical_Current_Test := 'REPROVADO';
       #Functional_Tests_Panels[25].Read_Electrical_Current := #In_Functional_Test_Odd.Electrical_Current_Read_PLC_Functional_Test_25;
   END_IF;
   IF #In_Functional_Test_Odd.Star_Test_PLC_Functional_Test_25 AND #In_Functional_Test_Odd.Electrical_Current_Test_Approved_PLC_Functional_Test_25 THEN
       #Functional_Tests_Panels[25].Electrical_Current_Test := 'APROVADO';
   END_IF;
   IF #In_Functional_Test_Odd.Star_Test_PLC_Functional_Test_25 AND #In_Functional_Test_Odd.Visual_Test_Approved_PLC_Functional_Test_25 THEN
       #Functional_Tests_Panels[25].Visual_Test := 'APROVADO';
   END_IF;
   IF #In_Functional_Test_Odd.Star_Test_PLC_Functional_Test_25 AND NOT #In_Functional_Test_Odd.Visual_Test_Approved_PLC_Functional_Test_25 THEN
       #Functional_Tests_Panels[25].Visual_Test := 'REPROVADO';
   END_IF;
   IF #In_Functional_Test_Odd.Star_Test_PLC_Functional_Test_25 AND #In_Functional_Test_Odd.Electrical_Current_Test_Approved_PLC_Functional_Test_25 AND #In_Functional_Test_Odd.Visual_Test_Approved_PLC_Functional_Test_25 THEN
       #Functional_Tests_Panels[25].Functional_Test := 'APROVADO';
   END_IF;
   IF #In_Functional_Test_Odd.Star_Test_PLC_Functional_Test_25 AND (NOT #In_Functional_Test_Odd.Electrical_Current_Test_Approved_PLC_Functional_Test_25 OR NOT #In_Functional_Test_Odd.Visual_Test_Approved_PLC_Functional_Test_25) THEN
       #Functional_Tests_Panels[25].Functional_Test := 'REPROVADO';
   END_IF;
END_REGION

REGION Network 26: Panel 26
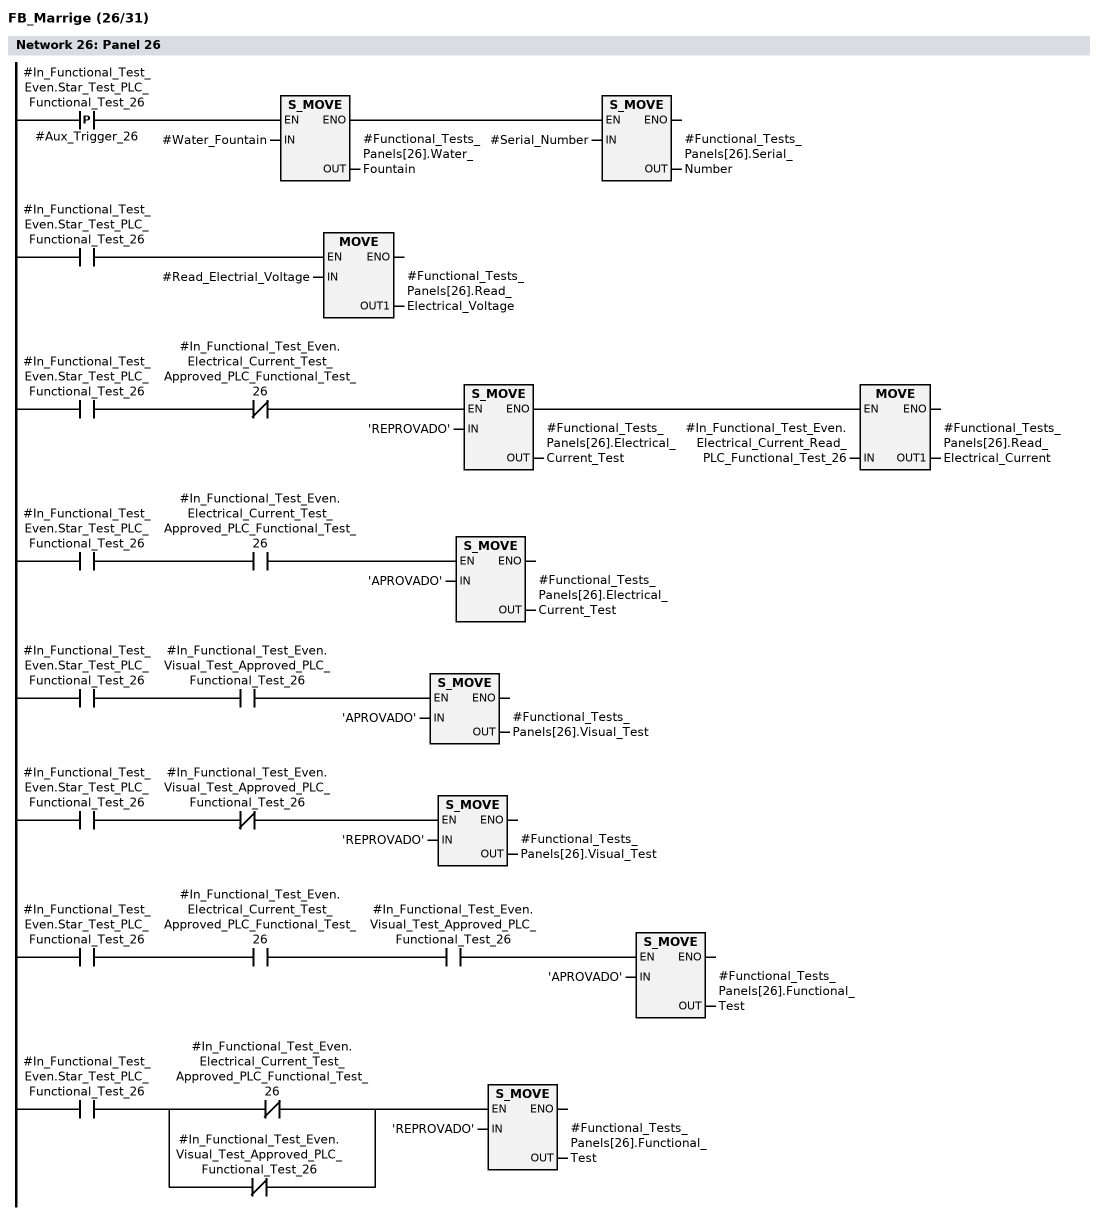
   RUNG wire#powerrail
      P_Contact(operand := #In_Functional_Test_Even.Star_Test_PLC_Functional_Test_26, bit := #Aux_Trigger_26)
      S_Move(in := #Water_Fountain, out => #Functional_Tests_Panels[26].Water_Fountain)
      S_Move(in := #Serial_Number, out => #Functional_Tests_Panels[26].Serial_Number)
   END_RUNG
   RUNG wire#powerrail
      Contact( #In_Functional_Test_Even.Star_Test_PLC_Functional_Test_26 )
      Move(in := #Read_Electrial_Voltage, out1 => #Functional_Tests_Panels[26].Read_Electrical_Voltage)
   END_RUNG
   RUNG wire#powerrail
      Contact( #In_Functional_Test_Even.Star_Test_PLC_Functional_Test_26 )
      I_Contact( #In_Functional_Test_Even.Electrical_Current_Test_Approved_PLC_Functional_Test_26 )
      S_Move(in := 'REPROVADO', out => #Functional_Tests_Panels[26].Electrical_Current_Test)
      Move(in := #In_Functional_Test_Even.Electrical_Current_Read_PLC_Functional_Test_26, out1 => #Functional_Tests_Panels[26].Read_Electrical_Current)
   END_RUNG
   RUNG wire#powerrail
      Contact( #In_Functional_Test_Even.Star_Test_PLC_Functional_Test_26 )
      Contact( #In_Functional_Test_Even.Electrical_Current_Test_Approved_PLC_Functional_Test_26 )
      S_Move(in := 'APROVADO', out => #Functional_Tests_Panels[26].Electrical_Current_Test)
   END_RUNG
   RUNG wire#powerrail
      Contact( #In_Functional_Test_Even.Star_Test_PLC_Functional_Test_26 )
      Contact( #In_Functional_Test_Even.Visual_Test_Approved_PLC_Functional_Test_26 )
      S_Move(in := 'APROVADO', out => #Functional_Tests_Panels[26].Visual_Test)
   END_RUNG
   RUNG wire#powerrail
      Contact( #In_Functional_Test_Even.Star_Test_PLC_Functional_Test_26 )
      I_Contact( #In_Functional_Test_Even.Visual_Test_Approved_PLC_Functional_Test_26 )
      S_Move(in := 'REPROVADO', out => #Functional_Tests_Panels[26].Visual_Test)
   END_RUNG
   RUNG wire#powerrail
      Contact( #In_Functional_Test_Even.Star_Test_PLC_Functional_Test_26 )
      Contact( #In_Functional_Test_Even.Electrical_Current_Test_Approved_PLC_Functional_Test_26 )
      Contact( #In_Functional_Test_Even.Visual_Test_Approved_PLC_Functional_Test_26 )
      S_Move(in := 'APROVADO', out => #Functional_Tests_Panels[26].Functional_Test)
   END_RUNG
   RUNG wire#powerrail
      Contact( #In_Functional_Test_Even.Star_Test_PLC_Functional_Test_26 )
      wire#w1
      I_Contact( #In_Functional_Test_Even.Electrical_Current_Test_Approved_PLC_Functional_Test_26 )
      wire#w2
      S_Move(in := 'REPROVADO', out => #Functional_Tests_Panels[26].Functional_Test)
   END_RUNG
   RUNG wire#w1
      I_Contact( #In_Functional_Test_Even.Visual_Test_Approved_PLC_Functional_Test_26 )
   END_RUNG wire#w2
   // the same network as SCL:
   #_w1 := #In_Functional_Test_Even.Star_Test_PLC_Functional_Test_26 AND NOT #Aux_Trigger_26;   // rising edge of #In_Functional_Test_Even.Star_Test_PLC_Functional_Test_26
   #Aux_Trigger_26 := #In_Functional_Test_Even.Star_Test_PLC_Functional_Test_26;
   IF #_w1 THEN
       #Functional_Tests_Panels[26].Water_Fountain := #Water_Fountain;
       #Functional_Tests_Panels[26].Serial_Number := #Serial_Number;
   END_IF;
   IF #In_Functional_Test_Even.Star_Test_PLC_Functional_Test_26 THEN
       #Functional_Tests_Panels[26].Read_Electrical_Voltage := #Read_Electrial_Voltage;
   END_IF;
   IF #In_Functional_Test_Even.Star_Test_PLC_Functional_Test_26 AND NOT #In_Functional_Test_Even.Electrical_Current_Test_Approved_PLC_Functional_Test_26 THEN
       #Functional_Tests_Panels[26].Electrical_Current_Test := 'REPROVADO';
       #Functional_Tests_Panels[26].Read_Electrical_Current := #In_Functional_Test_Even.Electrical_Current_Read_PLC_Functional_Test_26;
   END_IF;
   IF #In_Functional_Test_Even.Star_Test_PLC_Functional_Test_26 AND #In_Functional_Test_Even.Electrical_Current_Test_Approved_PLC_Functional_Test_26 THEN
       #Functional_Tests_Panels[26].Electrical_Current_Test := 'APROVADO';
   END_IF;
   IF #In_Functional_Test_Even.Star_Test_PLC_Functional_Test_26 AND #In_Functional_Test_Even.Visual_Test_Approved_PLC_Functional_Test_26 THEN
       #Functional_Tests_Panels[26].Visual_Test := 'APROVADO';
   END_IF;
   IF #In_Functional_Test_Even.Star_Test_PLC_Functional_Test_26 AND NOT #In_Functional_Test_Even.Visual_Test_Approved_PLC_Functional_Test_26 THEN
       #Functional_Tests_Panels[26].Visual_Test := 'REPROVADO';
   END_IF;
   IF #In_Functional_Test_Even.Star_Test_PLC_Functional_Test_26 AND #In_Functional_Test_Even.Electrical_Current_Test_Approved_PLC_Functional_Test_26 AND #In_Functional_Test_Even.Visual_Test_Approved_PLC_Functional_Test_26 THEN
       #Functional_Tests_Panels[26].Functional_Test := 'APROVADO';
   END_IF;
   IF #In_Functional_Test_Even.Star_Test_PLC_Functional_Test_26 AND (NOT #In_Functional_Test_Even.Electrical_Current_Test_Approved_PLC_Functional_Test_26 OR NOT #In_Functional_Test_Even.Visual_Test_Approved_PLC_Functional_Test_26) THEN
       #Functional_Tests_Panels[26].Functional_Test := 'REPROVADO';
   END_IF;
END_REGION

REGION Network 27: Panel 27
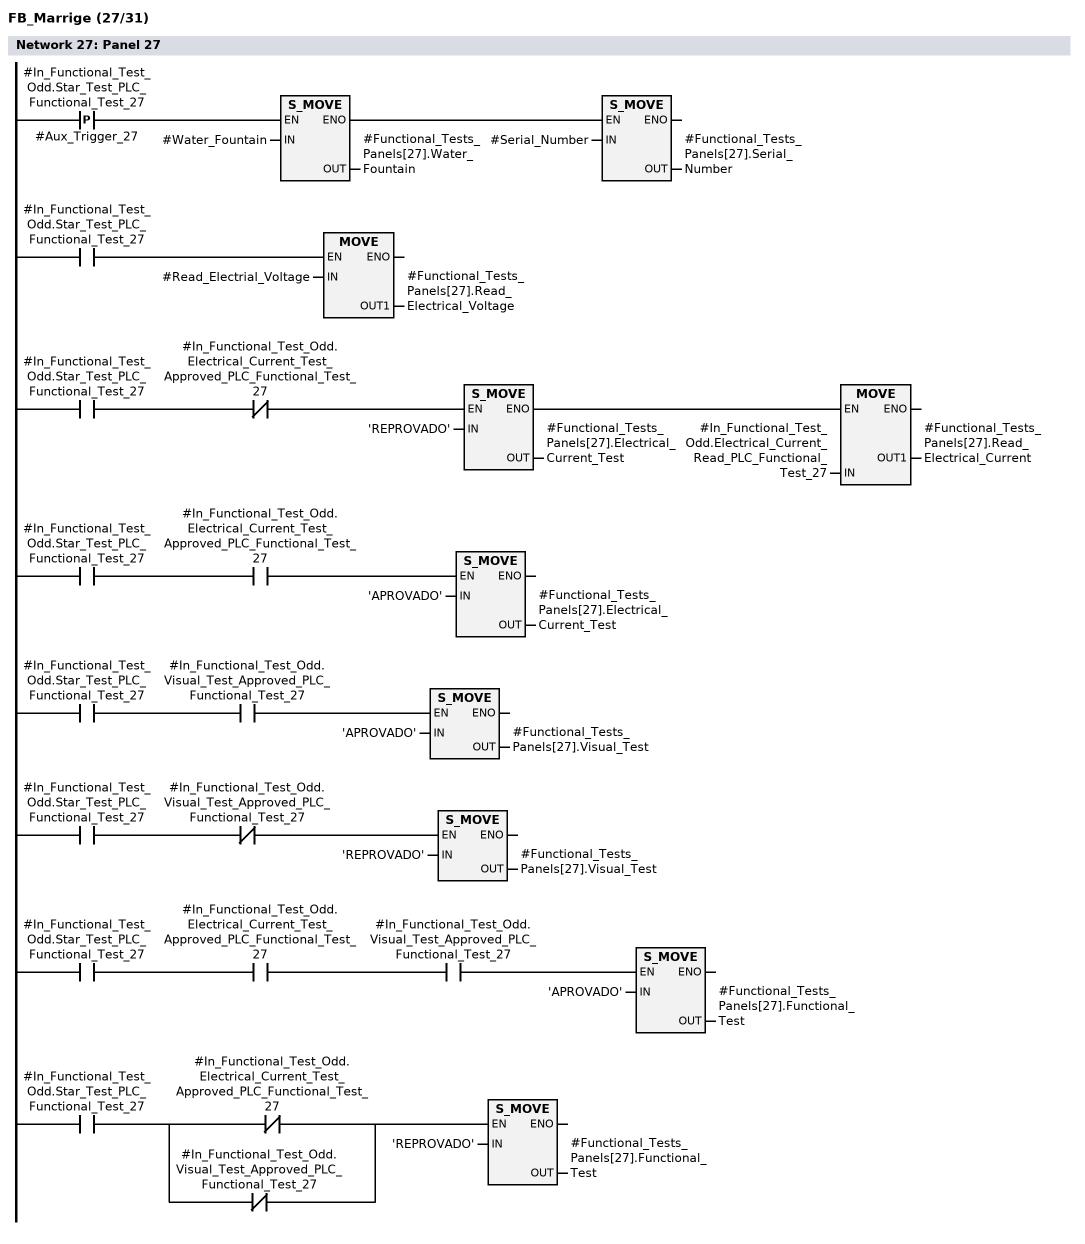
   RUNG wire#powerrail
      P_Contact(operand := #In_Functional_Test_Odd.Star_Test_PLC_Functional_Test_27, bit := #Aux_Trigger_27)
      S_Move(in := #Water_Fountain, out => #Functional_Tests_Panels[27].Water_Fountain)
      S_Move(in := #Serial_Number, out => #Functional_Tests_Panels[27].Serial_Number)
   END_RUNG
   RUNG wire#powerrail
      Contact( #In_Functional_Test_Odd.Star_Test_PLC_Functional_Test_27 )
      Move(in := #Read_Electrial_Voltage, out1 => #Functional_Tests_Panels[27].Read_Electrical_Voltage)
   END_RUNG
   RUNG wire#powerrail
      Contact( #In_Functional_Test_Odd.Star_Test_PLC_Functional_Test_27 )
      I_Contact( #In_Functional_Test_Odd.Electrical_Current_Test_Approved_PLC_Functional_Test_27 )
      S_Move(in := 'REPROVADO', out => #Functional_Tests_Panels[27].Electrical_Current_Test)
      Move(in := #In_Functional_Test_Odd.Electrical_Current_Read_PLC_Functional_Test_27, out1 => #Functional_Tests_Panels[27].Read_Electrical_Current)
   END_RUNG
   RUNG wire#powerrail
      Contact( #In_Functional_Test_Odd.Star_Test_PLC_Functional_Test_27 )
      Contact( #In_Functional_Test_Odd.Electrical_Current_Test_Approved_PLC_Functional_Test_27 )
      S_Move(in := 'APROVADO', out => #Functional_Tests_Panels[27].Electrical_Current_Test)
   END_RUNG
   RUNG wire#powerrail
      Contact( #In_Functional_Test_Odd.Star_Test_PLC_Functional_Test_27 )
      Contact( #In_Functional_Test_Odd.Visual_Test_Approved_PLC_Functional_Test_27 )
      S_Move(in := 'APROVADO', out => #Functional_Tests_Panels[27].Visual_Test)
   END_RUNG
   RUNG wire#powerrail
      Contact( #In_Functional_Test_Odd.Star_Test_PLC_Functional_Test_27 )
      I_Contact( #In_Functional_Test_Odd.Visual_Test_Approved_PLC_Functional_Test_27 )
      S_Move(in := 'REPROVADO', out => #Functional_Tests_Panels[27].Visual_Test)
   END_RUNG
   RUNG wire#powerrail
      Contact( #In_Functional_Test_Odd.Star_Test_PLC_Functional_Test_27 )
      Contact( #In_Functional_Test_Odd.Electrical_Current_Test_Approved_PLC_Functional_Test_27 )
      Contact( #In_Functional_Test_Odd.Visual_Test_Approved_PLC_Functional_Test_27 )
      S_Move(in := 'APROVADO', out => #Functional_Tests_Panels[27].Functional_Test)
   END_RUNG
   RUNG wire#powerrail
      Contact( #In_Functional_Test_Odd.Star_Test_PLC_Functional_Test_27 )
      wire#w1
      I_Contact( #In_Functional_Test_Odd.Electrical_Current_Test_Approved_PLC_Functional_Test_27 )
      wire#w2
      S_Move(in := 'REPROVADO', out => #Functional_Tests_Panels[27].Functional_Test)
   END_RUNG
   RUNG wire#w1
      I_Contact( #In_Functional_Test_Odd.Visual_Test_Approved_PLC_Functional_Test_27 )
   END_RUNG wire#w2
   // the same network as SCL:
   #_w1 := #In_Functional_Test_Odd.Star_Test_PLC_Functional_Test_27 AND NOT #Aux_Trigger_27;   // rising edge of #In_Functional_Test_Odd.Star_Test_PLC_Functional_Test_27
   #Aux_Trigger_27 := #In_Functional_Test_Odd.Star_Test_PLC_Functional_Test_27;
   IF #_w1 THEN
       #Functional_Tests_Panels[27].Water_Fountain := #Water_Fountain;
       #Functional_Tests_Panels[27].Serial_Number := #Serial_Number;
   END_IF;
   IF #In_Functional_Test_Odd.Star_Test_PLC_Functional_Test_27 THEN
       #Functional_Tests_Panels[27].Read_Electrical_Voltage := #Read_Electrial_Voltage;
   END_IF;
   IF #In_Functional_Test_Odd.Star_Test_PLC_Functional_Test_27 AND NOT #In_Functional_Test_Odd.Electrical_Current_Test_Approved_PLC_Functional_Test_27 THEN
       #Functional_Tests_Panels[27].Electrical_Current_Test := 'REPROVADO';
       #Functional_Tests_Panels[27].Read_Electrical_Current := #In_Functional_Test_Odd.Electrical_Current_Read_PLC_Functional_Test_27;
   END_IF;
   IF #In_Functional_Test_Odd.Star_Test_PLC_Functional_Test_27 AND #In_Functional_Test_Odd.Electrical_Current_Test_Approved_PLC_Functional_Test_27 THEN
       #Functional_Tests_Panels[27].Electrical_Current_Test := 'APROVADO';
   END_IF;
   IF #In_Functional_Test_Odd.Star_Test_PLC_Functional_Test_27 AND #In_Functional_Test_Odd.Visual_Test_Approved_PLC_Functional_Test_27 THEN
       #Functional_Tests_Panels[27].Visual_Test := 'APROVADO';
   END_IF;
   IF #In_Functional_Test_Odd.Star_Test_PLC_Functional_Test_27 AND NOT #In_Functional_Test_Odd.Visual_Test_Approved_PLC_Functional_Test_27 THEN
       #Functional_Tests_Panels[27].Visual_Test := 'REPROVADO';
   END_IF;
   IF #In_Functional_Test_Odd.Star_Test_PLC_Functional_Test_27 AND #In_Functional_Test_Odd.Electrical_Current_Test_Approved_PLC_Functional_Test_27 AND #In_Functional_Test_Odd.Visual_Test_Approved_PLC_Functional_Test_27 THEN
       #Functional_Tests_Panels[27].Functional_Test := 'APROVADO';
   END_IF;
   IF #In_Functional_Test_Odd.Star_Test_PLC_Functional_Test_27 AND (NOT #In_Functional_Test_Odd.Electrical_Current_Test_Approved_PLC_Functional_Test_27 OR NOT #In_Functional_Test_Odd.Visual_Test_Approved_PLC_Functional_Test_27) THEN
       #Functional_Tests_Panels[27].Functional_Test := 'REPROVADO';
   END_IF;
END_REGION

REGION Network 28: Panel 28
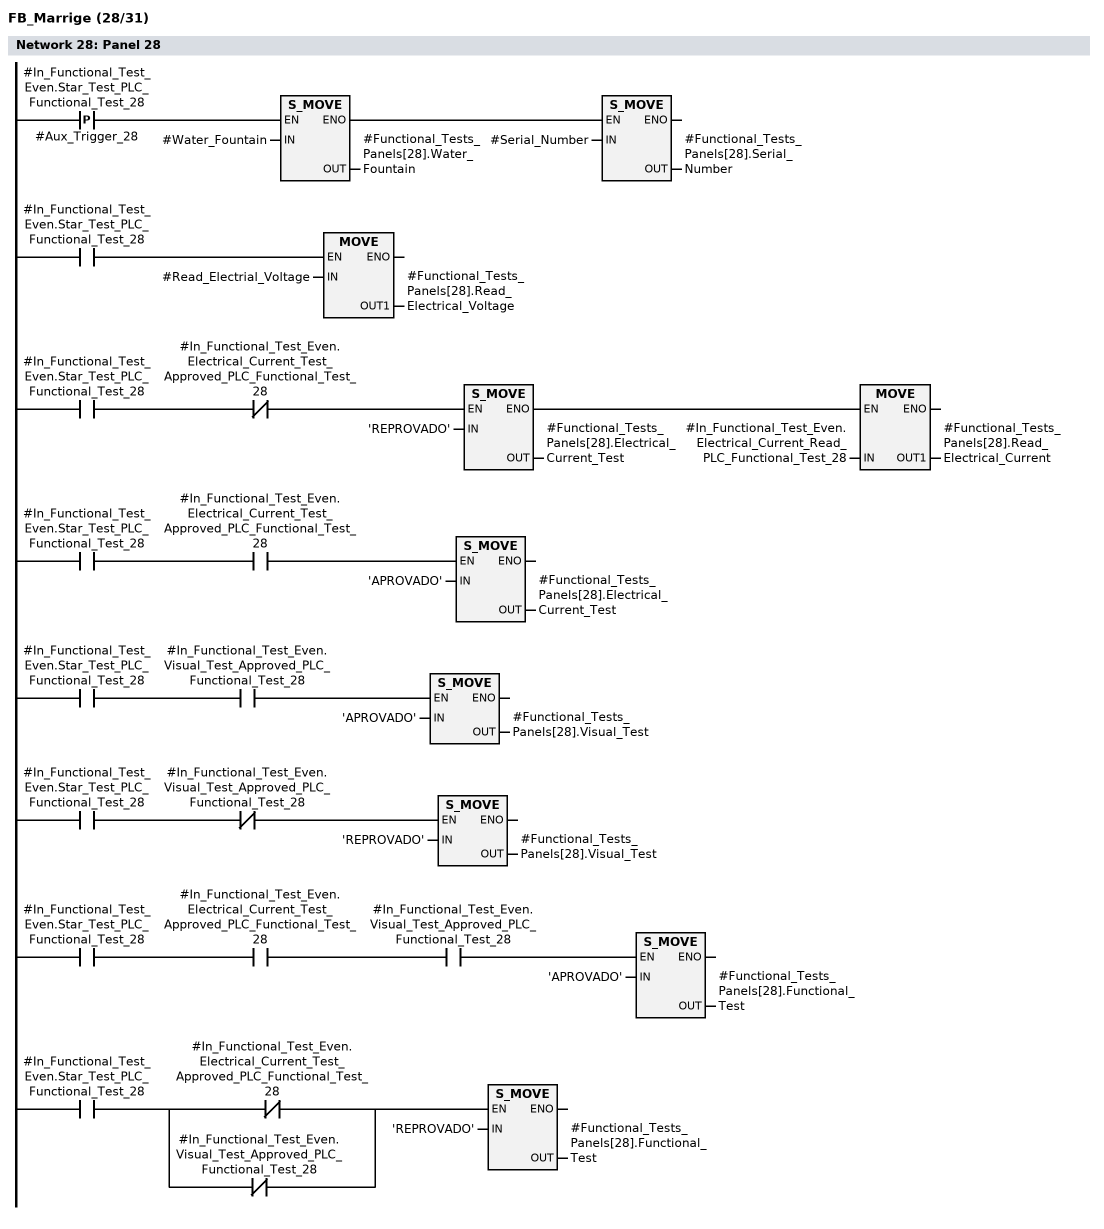
   RUNG wire#powerrail
      P_Contact(operand := #In_Functional_Test_Even.Star_Test_PLC_Functional_Test_28, bit := #Aux_Trigger_28)
      S_Move(in := #Water_Fountain, out => #Functional_Tests_Panels[28].Water_Fountain)
      S_Move(in := #Serial_Number, out => #Functional_Tests_Panels[28].Serial_Number)
   END_RUNG
   RUNG wire#powerrail
      Contact( #In_Functional_Test_Even.Star_Test_PLC_Functional_Test_28 )
      Move(in := #Read_Electrial_Voltage, out1 => #Functional_Tests_Panels[28].Read_Electrical_Voltage)
   END_RUNG
   RUNG wire#powerrail
      Contact( #In_Functional_Test_Even.Star_Test_PLC_Functional_Test_28 )
      I_Contact( #In_Functional_Test_Even.Electrical_Current_Test_Approved_PLC_Functional_Test_28 )
      S_Move(in := 'REPROVADO', out => #Functional_Tests_Panels[28].Electrical_Current_Test)
      Move(in := #In_Functional_Test_Even.Electrical_Current_Read_PLC_Functional_Test_28, out1 => #Functional_Tests_Panels[28].Read_Electrical_Current)
   END_RUNG
   RUNG wire#powerrail
      Contact( #In_Functional_Test_Even.Star_Test_PLC_Functional_Test_28 )
      Contact( #In_Functional_Test_Even.Electrical_Current_Test_Approved_PLC_Functional_Test_28 )
      S_Move(in := 'APROVADO', out => #Functional_Tests_Panels[28].Electrical_Current_Test)
   END_RUNG
   RUNG wire#powerrail
      Contact( #In_Functional_Test_Even.Star_Test_PLC_Functional_Test_28 )
      Contact( #In_Functional_Test_Even.Visual_Test_Approved_PLC_Functional_Test_28 )
      S_Move(in := 'APROVADO', out => #Functional_Tests_Panels[28].Visual_Test)
   END_RUNG
   RUNG wire#powerrail
      Contact( #In_Functional_Test_Even.Star_Test_PLC_Functional_Test_28 )
      I_Contact( #In_Functional_Test_Even.Visual_Test_Approved_PLC_Functional_Test_28 )
      S_Move(in := 'REPROVADO', out => #Functional_Tests_Panels[28].Visual_Test)
   END_RUNG
   RUNG wire#powerrail
      Contact( #In_Functional_Test_Even.Star_Test_PLC_Functional_Test_28 )
      Contact( #In_Functional_Test_Even.Electrical_Current_Test_Approved_PLC_Functional_Test_28 )
      Contact( #In_Functional_Test_Even.Visual_Test_Approved_PLC_Functional_Test_28 )
      S_Move(in := 'APROVADO', out => #Functional_Tests_Panels[28].Functional_Test)
   END_RUNG
   RUNG wire#powerrail
      Contact( #In_Functional_Test_Even.Star_Test_PLC_Functional_Test_28 )
      wire#w1
      I_Contact( #In_Functional_Test_Even.Electrical_Current_Test_Approved_PLC_Functional_Test_28 )
      wire#w2
      S_Move(in := 'REPROVADO', out => #Functional_Tests_Panels[28].Functional_Test)
   END_RUNG
   RUNG wire#w1
      I_Contact( #In_Functional_Test_Even.Visual_Test_Approved_PLC_Functional_Test_28 )
   END_RUNG wire#w2
   // the same network as SCL:
   #_w1 := #In_Functional_Test_Even.Star_Test_PLC_Functional_Test_28 AND NOT #Aux_Trigger_28;   // rising edge of #In_Functional_Test_Even.Star_Test_PLC_Functional_Test_28
   #Aux_Trigger_28 := #In_Functional_Test_Even.Star_Test_PLC_Functional_Test_28;
   IF #_w1 THEN
       #Functional_Tests_Panels[28].Water_Fountain := #Water_Fountain;
       #Functional_Tests_Panels[28].Serial_Number := #Serial_Number;
   END_IF;
   IF #In_Functional_Test_Even.Star_Test_PLC_Functional_Test_28 THEN
       #Functional_Tests_Panels[28].Read_Electrical_Voltage := #Read_Electrial_Voltage;
   END_IF;
   IF #In_Functional_Test_Even.Star_Test_PLC_Functional_Test_28 AND NOT #In_Functional_Test_Even.Electrical_Current_Test_Approved_PLC_Functional_Test_28 THEN
       #Functional_Tests_Panels[28].Electrical_Current_Test := 'REPROVADO';
       #Functional_Tests_Panels[28].Read_Electrical_Current := #In_Functional_Test_Even.Electrical_Current_Read_PLC_Functional_Test_28;
   END_IF;
   IF #In_Functional_Test_Even.Star_Test_PLC_Functional_Test_28 AND #In_Functional_Test_Even.Electrical_Current_Test_Approved_PLC_Functional_Test_28 THEN
       #Functional_Tests_Panels[28].Electrical_Current_Test := 'APROVADO';
   END_IF;
   IF #In_Functional_Test_Even.Star_Test_PLC_Functional_Test_28 AND #In_Functional_Test_Even.Visual_Test_Approved_PLC_Functional_Test_28 THEN
       #Functional_Tests_Panels[28].Visual_Test := 'APROVADO';
   END_IF;
   IF #In_Functional_Test_Even.Star_Test_PLC_Functional_Test_28 AND NOT #In_Functional_Test_Even.Visual_Test_Approved_PLC_Functional_Test_28 THEN
       #Functional_Tests_Panels[28].Visual_Test := 'REPROVADO';
   END_IF;
   IF #In_Functional_Test_Even.Star_Test_PLC_Functional_Test_28 AND #In_Functional_Test_Even.Electrical_Current_Test_Approved_PLC_Functional_Test_28 AND #In_Functional_Test_Even.Visual_Test_Approved_PLC_Functional_Test_28 THEN
       #Functional_Tests_Panels[28].Functional_Test := 'APROVADO';
   END_IF;
   IF #In_Functional_Test_Even.Star_Test_PLC_Functional_Test_28 AND (NOT #In_Functional_Test_Even.Electrical_Current_Test_Approved_PLC_Functional_Test_28 OR NOT #In_Functional_Test_Even.Visual_Test_Approved_PLC_Functional_Test_28) THEN
       #Functional_Tests_Panels[28].Functional_Test := 'REPROVADO';
   END_IF;
END_REGION

REGION Network 29: Panel 29
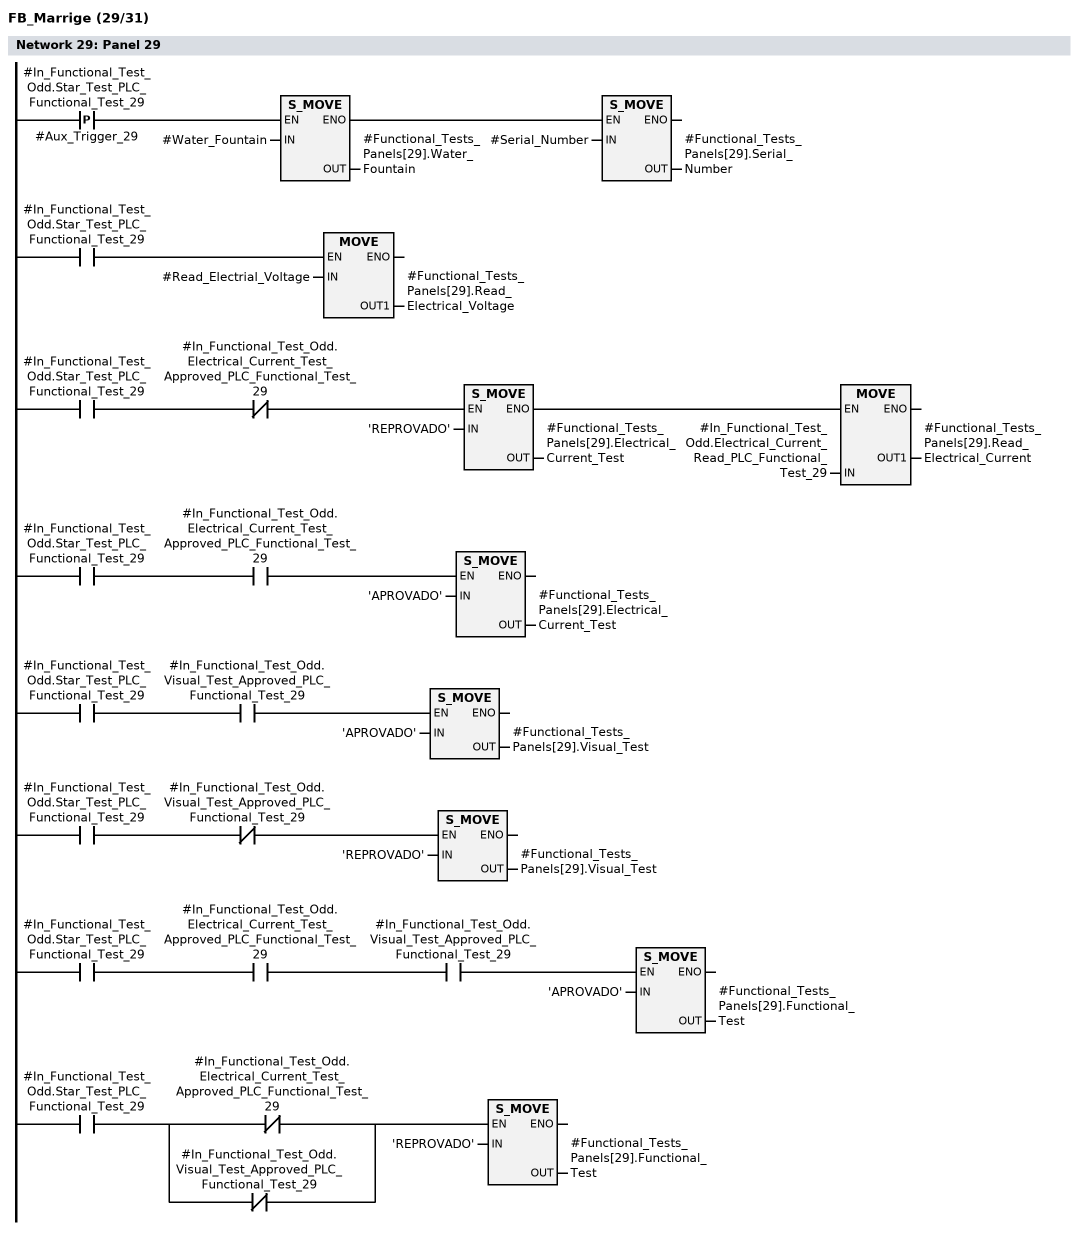
   RUNG wire#powerrail
      P_Contact(operand := #In_Functional_Test_Odd.Star_Test_PLC_Functional_Test_29, bit := #Aux_Trigger_29)
      S_Move(in := #Water_Fountain, out => #Functional_Tests_Panels[29].Water_Fountain)
      S_Move(in := #Serial_Number, out => #Functional_Tests_Panels[29].Serial_Number)
   END_RUNG
   RUNG wire#powerrail
      Contact( #In_Functional_Test_Odd.Star_Test_PLC_Functional_Test_29 )
      Move(in := #Read_Electrial_Voltage, out1 => #Functional_Tests_Panels[29].Read_Electrical_Voltage)
   END_RUNG
   RUNG wire#powerrail
      Contact( #In_Functional_Test_Odd.Star_Test_PLC_Functional_Test_29 )
      I_Contact( #In_Functional_Test_Odd.Electrical_Current_Test_Approved_PLC_Functional_Test_29 )
      S_Move(in := 'REPROVADO', out => #Functional_Tests_Panels[29].Electrical_Current_Test)
      Move(in := #In_Functional_Test_Odd.Electrical_Current_Read_PLC_Functional_Test_29, out1 => #Functional_Tests_Panels[29].Read_Electrical_Current)
   END_RUNG
   RUNG wire#powerrail
      Contact( #In_Functional_Test_Odd.Star_Test_PLC_Functional_Test_29 )
      Contact( #In_Functional_Test_Odd.Electrical_Current_Test_Approved_PLC_Functional_Test_29 )
      S_Move(in := 'APROVADO', out => #Functional_Tests_Panels[29].Electrical_Current_Test)
   END_RUNG
   RUNG wire#powerrail
      Contact( #In_Functional_Test_Odd.Star_Test_PLC_Functional_Test_29 )
      Contact( #In_Functional_Test_Odd.Visual_Test_Approved_PLC_Functional_Test_29 )
      S_Move(in := 'APROVADO', out => #Functional_Tests_Panels[29].Visual_Test)
   END_RUNG
   RUNG wire#powerrail
      Contact( #In_Functional_Test_Odd.Star_Test_PLC_Functional_Test_29 )
      I_Contact( #In_Functional_Test_Odd.Visual_Test_Approved_PLC_Functional_Test_29 )
      S_Move(in := 'REPROVADO', out => #Functional_Tests_Panels[29].Visual_Test)
   END_RUNG
   RUNG wire#powerrail
      Contact( #In_Functional_Test_Odd.Star_Test_PLC_Functional_Test_29 )
      Contact( #In_Functional_Test_Odd.Electrical_Current_Test_Approved_PLC_Functional_Test_29 )
      Contact( #In_Functional_Test_Odd.Visual_Test_Approved_PLC_Functional_Test_29 )
      S_Move(in := 'APROVADO', out => #Functional_Tests_Panels[29].Functional_Test)
   END_RUNG
   RUNG wire#powerrail
      Contact( #In_Functional_Test_Odd.Star_Test_PLC_Functional_Test_29 )
      wire#w1
      I_Contact( #In_Functional_Test_Odd.Electrical_Current_Test_Approved_PLC_Functional_Test_29 )
      wire#w2
      S_Move(in := 'REPROVADO', out => #Functional_Tests_Panels[29].Functional_Test)
   END_RUNG
   RUNG wire#w1
      I_Contact( #In_Functional_Test_Odd.Visual_Test_Approved_PLC_Functional_Test_29 )
   END_RUNG wire#w2
   // the same network as SCL:
   #_w1 := #In_Functional_Test_Odd.Star_Test_PLC_Functional_Test_29 AND NOT #Aux_Trigger_29;   // rising edge of #In_Functional_Test_Odd.Star_Test_PLC_Functional_Test_29
   #Aux_Trigger_29 := #In_Functional_Test_Odd.Star_Test_PLC_Functional_Test_29;
   IF #_w1 THEN
       #Functional_Tests_Panels[29].Water_Fountain := #Water_Fountain;
       #Functional_Tests_Panels[29].Serial_Number := #Serial_Number;
   END_IF;
   IF #In_Functional_Test_Odd.Star_Test_PLC_Functional_Test_29 THEN
       #Functional_Tests_Panels[29].Read_Electrical_Voltage := #Read_Electrial_Voltage;
   END_IF;
   IF #In_Functional_Test_Odd.Star_Test_PLC_Functional_Test_29 AND NOT #In_Functional_Test_Odd.Electrical_Current_Test_Approved_PLC_Functional_Test_29 THEN
       #Functional_Tests_Panels[29].Electrical_Current_Test := 'REPROVADO';
       #Functional_Tests_Panels[29].Read_Electrical_Current := #In_Functional_Test_Odd.Electrical_Current_Read_PLC_Functional_Test_29;
   END_IF;
   IF #In_Functional_Test_Odd.Star_Test_PLC_Functional_Test_29 AND #In_Functional_Test_Odd.Electrical_Current_Test_Approved_PLC_Functional_Test_29 THEN
       #Functional_Tests_Panels[29].Electrical_Current_Test := 'APROVADO';
   END_IF;
   IF #In_Functional_Test_Odd.Star_Test_PLC_Functional_Test_29 AND #In_Functional_Test_Odd.Visual_Test_Approved_PLC_Functional_Test_29 THEN
       #Functional_Tests_Panels[29].Visual_Test := 'APROVADO';
   END_IF;
   IF #In_Functional_Test_Odd.Star_Test_PLC_Functional_Test_29 AND NOT #In_Functional_Test_Odd.Visual_Test_Approved_PLC_Functional_Test_29 THEN
       #Functional_Tests_Panels[29].Visual_Test := 'REPROVADO';
   END_IF;
   IF #In_Functional_Test_Odd.Star_Test_PLC_Functional_Test_29 AND #In_Functional_Test_Odd.Electrical_Current_Test_Approved_PLC_Functional_Test_29 AND #In_Functional_Test_Odd.Visual_Test_Approved_PLC_Functional_Test_29 THEN
       #Functional_Tests_Panels[29].Functional_Test := 'APROVADO';
   END_IF;
   IF #In_Functional_Test_Odd.Star_Test_PLC_Functional_Test_29 AND (NOT #In_Functional_Test_Odd.Electrical_Current_Test_Approved_PLC_Functional_Test_29 OR NOT #In_Functional_Test_Odd.Visual_Test_Approved_PLC_Functional_Test_29) THEN
       #Functional_Tests_Panels[29].Functional_Test := 'REPROVADO';
   END_IF;
END_REGION

REGION Network 30: Panel 30
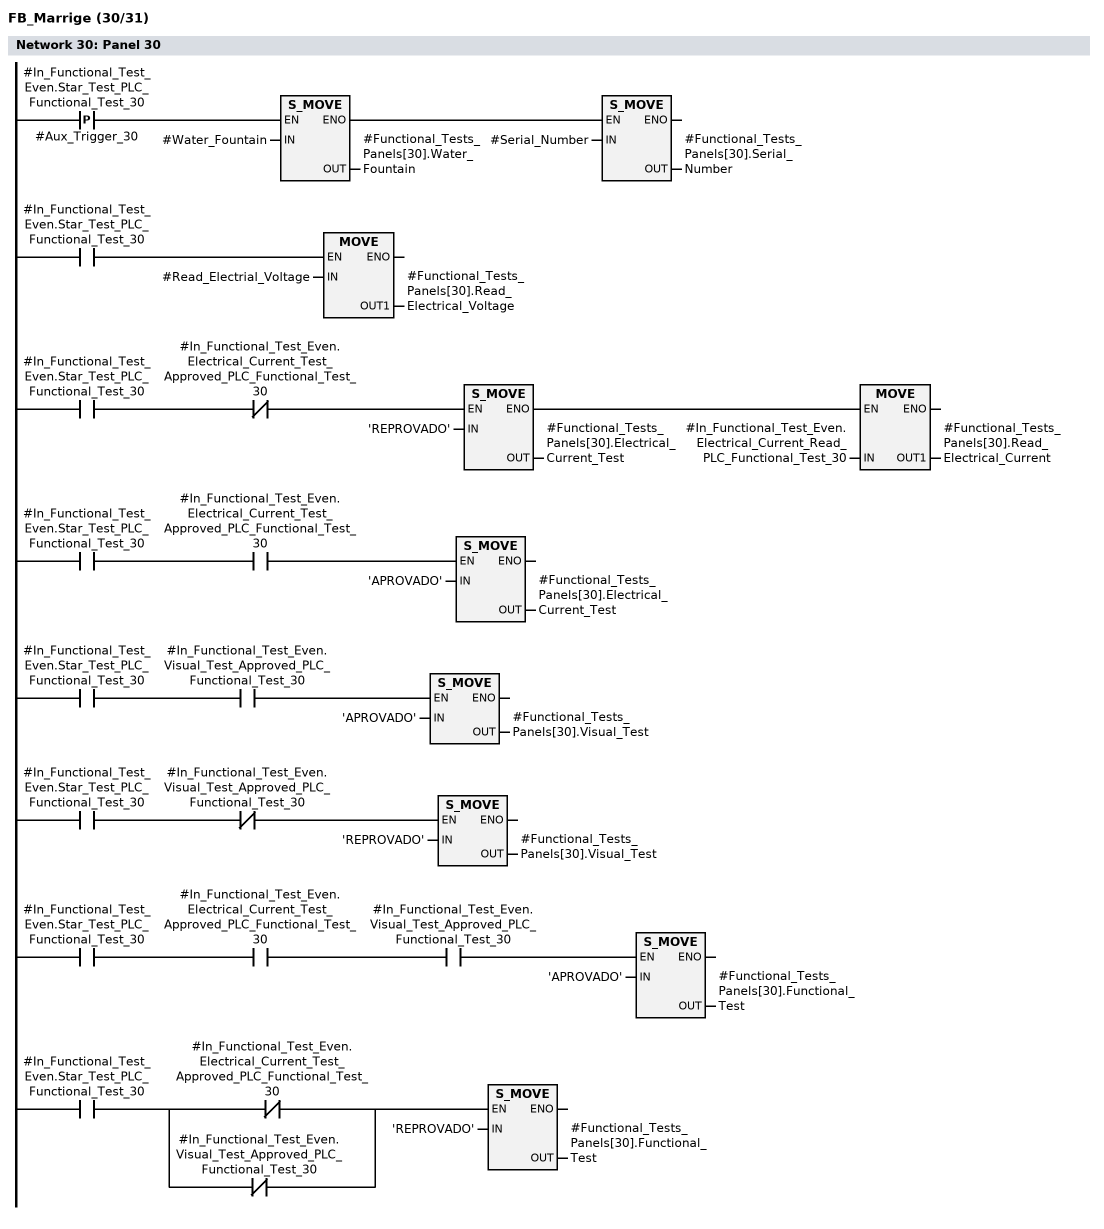
   RUNG wire#powerrail
      P_Contact(operand := #In_Functional_Test_Even.Star_Test_PLC_Functional_Test_30, bit := #Aux_Trigger_30)
      S_Move(in := #Water_Fountain, out => #Functional_Tests_Panels[30].Water_Fountain)
      S_Move(in := #Serial_Number, out => #Functional_Tests_Panels[30].Serial_Number)
   END_RUNG
   RUNG wire#powerrail
      Contact( #In_Functional_Test_Even.Star_Test_PLC_Functional_Test_30 )
      Move(in := #Read_Electrial_Voltage, out1 => #Functional_Tests_Panels[30].Read_Electrical_Voltage)
   END_RUNG
   RUNG wire#powerrail
      Contact( #In_Functional_Test_Even.Star_Test_PLC_Functional_Test_30 )
      I_Contact( #In_Functional_Test_Even.Electrical_Current_Test_Approved_PLC_Functional_Test_30 )
      S_Move(in := 'REPROVADO', out => #Functional_Tests_Panels[30].Electrical_Current_Test)
      Move(in := #In_Functional_Test_Even.Electrical_Current_Read_PLC_Functional_Test_30, out1 => #Functional_Tests_Panels[30].Read_Electrical_Current)
   END_RUNG
   RUNG wire#powerrail
      Contact( #In_Functional_Test_Even.Star_Test_PLC_Functional_Test_30 )
      Contact( #In_Functional_Test_Even.Electrical_Current_Test_Approved_PLC_Functional_Test_30 )
      S_Move(in := 'APROVADO', out => #Functional_Tests_Panels[30].Electrical_Current_Test)
   END_RUNG
   RUNG wire#powerrail
      Contact( #In_Functional_Test_Even.Star_Test_PLC_Functional_Test_30 )
      Contact( #In_Functional_Test_Even.Visual_Test_Approved_PLC_Functional_Test_30 )
      S_Move(in := 'APROVADO', out => #Functional_Tests_Panels[30].Visual_Test)
   END_RUNG
   RUNG wire#powerrail
      Contact( #In_Functional_Test_Even.Star_Test_PLC_Functional_Test_30 )
      I_Contact( #In_Functional_Test_Even.Visual_Test_Approved_PLC_Functional_Test_30 )
      S_Move(in := 'REPROVADO', out => #Functional_Tests_Panels[30].Visual_Test)
   END_RUNG
   RUNG wire#powerrail
      Contact( #In_Functional_Test_Even.Star_Test_PLC_Functional_Test_30 )
      Contact( #In_Functional_Test_Even.Electrical_Current_Test_Approved_PLC_Functional_Test_30 )
      Contact( #In_Functional_Test_Even.Visual_Test_Approved_PLC_Functional_Test_30 )
      S_Move(in := 'APROVADO', out => #Functional_Tests_Panels[30].Functional_Test)
   END_RUNG
   RUNG wire#powerrail
      Contact( #In_Functional_Test_Even.Star_Test_PLC_Functional_Test_30 )
      wire#w1
      I_Contact( #In_Functional_Test_Even.Electrical_Current_Test_Approved_PLC_Functional_Test_30 )
      wire#w2
      S_Move(in := 'REPROVADO', out => #Functional_Tests_Panels[30].Functional_Test)
   END_RUNG
   RUNG wire#w1
      I_Contact( #In_Functional_Test_Even.Visual_Test_Approved_PLC_Functional_Test_30 )
   END_RUNG wire#w2
   // the same network as SCL:
   #_w1 := #In_Functional_Test_Even.Star_Test_PLC_Functional_Test_30 AND NOT #Aux_Trigger_30;   // rising edge of #In_Functional_Test_Even.Star_Test_PLC_Functional_Test_30
   #Aux_Trigger_30 := #In_Functional_Test_Even.Star_Test_PLC_Functional_Test_30;
   IF #_w1 THEN
       #Functional_Tests_Panels[30].Water_Fountain := #Water_Fountain;
       #Functional_Tests_Panels[30].Serial_Number := #Serial_Number;
   END_IF;
   IF #In_Functional_Test_Even.Star_Test_PLC_Functional_Test_30 THEN
       #Functional_Tests_Panels[30].Read_Electrical_Voltage := #Read_Electrial_Voltage;
   END_IF;
   IF #In_Functional_Test_Even.Star_Test_PLC_Functional_Test_30 AND NOT #In_Functional_Test_Even.Electrical_Current_Test_Approved_PLC_Functional_Test_30 THEN
       #Functional_Tests_Panels[30].Electrical_Current_Test := 'REPROVADO';
       #Functional_Tests_Panels[30].Read_Electrical_Current := #In_Functional_Test_Even.Electrical_Current_Read_PLC_Functional_Test_30;
   END_IF;
   IF #In_Functional_Test_Even.Star_Test_PLC_Functional_Test_30 AND #In_Functional_Test_Even.Electrical_Current_Test_Approved_PLC_Functional_Test_30 THEN
       #Functional_Tests_Panels[30].Electrical_Current_Test := 'APROVADO';
   END_IF;
   IF #In_Functional_Test_Even.Star_Test_PLC_Functional_Test_30 AND #In_Functional_Test_Even.Visual_Test_Approved_PLC_Functional_Test_30 THEN
       #Functional_Tests_Panels[30].Visual_Test := 'APROVADO';
   END_IF;
   IF #In_Functional_Test_Even.Star_Test_PLC_Functional_Test_30 AND NOT #In_Functional_Test_Even.Visual_Test_Approved_PLC_Functional_Test_30 THEN
       #Functional_Tests_Panels[30].Visual_Test := 'REPROVADO';
   END_IF;
   IF #In_Functional_Test_Even.Star_Test_PLC_Functional_Test_30 AND #In_Functional_Test_Even.Electrical_Current_Test_Approved_PLC_Functional_Test_30 AND #In_Functional_Test_Even.Visual_Test_Approved_PLC_Functional_Test_30 THEN
       #Functional_Tests_Panels[30].Functional_Test := 'APROVADO';
   END_IF;
   IF #In_Functional_Test_Even.Star_Test_PLC_Functional_Test_30 AND (NOT #In_Functional_Test_Even.Electrical_Current_Test_Approved_PLC_Functional_Test_30 OR NOT #In_Functional_Test_Even.Visual_Test_Approved_PLC_Functional_Test_30) THEN
       #Functional_Tests_Panels[30].Functional_Test := 'REPROVADO';
   END_IF;
END_REGION

REGION Network 31: Got married
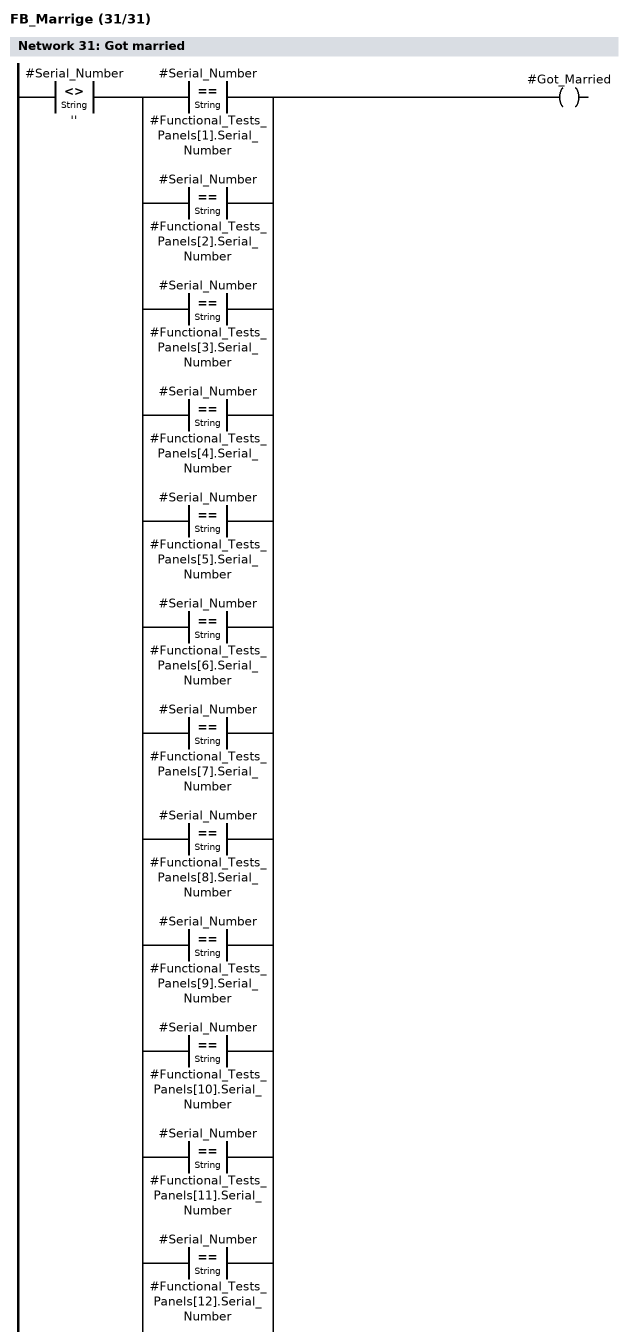
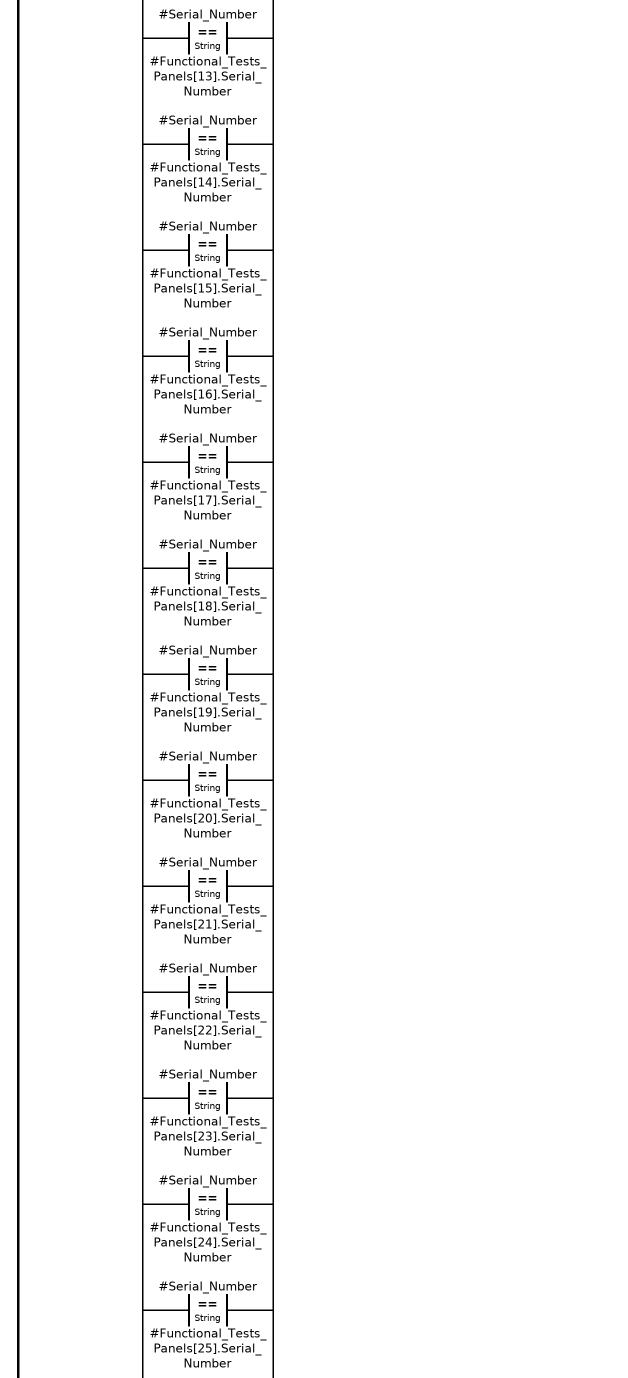
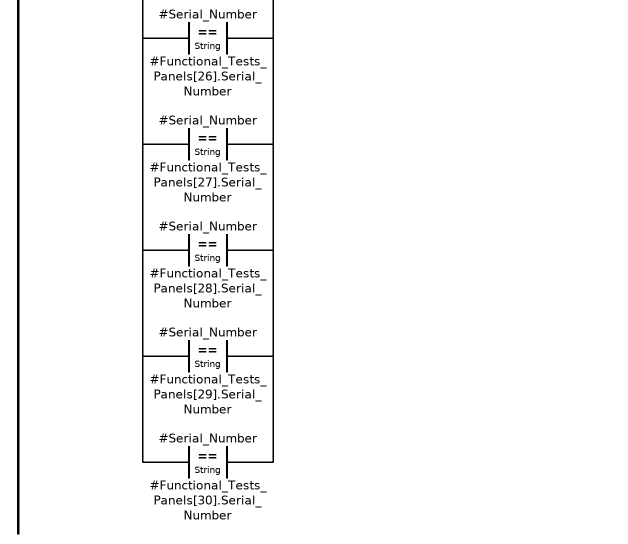
   RUNG wire#powerrail
      { S7_Templates := "SrcType := String" } NE_Contact(in1 := #Serial_Number, in2 := '')
      wire#w1
      { S7_Templates := "SrcType := String" } EQ_Contact(in1 := #Serial_Number, in2 := #Functional_Tests_Panels[1].Serial_Number)
      wire#w2
      Coil( #Got_Married )
   END_RUNG
   RUNG wire#w1
      { S7_Templates := "SrcType := String" } EQ_Contact(in1 := #Serial_Number, in2 := #Functional_Tests_Panels[2].Serial_Number)
   END_RUNG wire#w2
   RUNG wire#w1
      { S7_Templates := "SrcType := String" } EQ_Contact(in1 := #Serial_Number, in2 := #Functional_Tests_Panels[3].Serial_Number)
   END_RUNG wire#w2
   RUNG wire#w1
      { S7_Templates := "SrcType := String" } EQ_Contact(in1 := #Serial_Number, in2 := #Functional_Tests_Panels[4].Serial_Number)
   END_RUNG wire#w2
   RUNG wire#w1
      { S7_Templates := "SrcType := String" } EQ_Contact(in1 := #Serial_Number, in2 := #Functional_Tests_Panels[5].Serial_Number)
   END_RUNG wire#w2
   RUNG wire#w1
      { S7_Templates := "SrcType := String" } EQ_Contact(in1 := #Serial_Number, in2 := #Functional_Tests_Panels[6].Serial_Number)
   END_RUNG wire#w2
   RUNG wire#w1
      { S7_Templates := "SrcType := String" } EQ_Contact(in1 := #Serial_Number, in2 := #Functional_Tests_Panels[7].Serial_Number)
   END_RUNG wire#w2
   RUNG wire#w1
      { S7_Templates := "SrcType := String" } EQ_Contact(in1 := #Serial_Number, in2 := #Functional_Tests_Panels[8].Serial_Number)
   END_RUNG wire#w2
   RUNG wire#w1
      { S7_Templates := "SrcType := String" } EQ_Contact(in1 := #Serial_Number, in2 := #Functional_Tests_Panels[9].Serial_Number)
   END_RUNG wire#w2
   RUNG wire#w1
      { S7_Templates := "SrcType := String" } EQ_Contact(in1 := #Serial_Number, in2 := #Functional_Tests_Panels[10].Serial_Number)
   END_RUNG wire#w2
   RUNG wire#w1
      { S7_Templates := "SrcType := String" } EQ_Contact(in1 := #Serial_Number, in2 := #Functional_Tests_Panels[11].Serial_Number)
   END_RUNG wire#w2
   RUNG wire#w1
      { S7_Templates := "SrcType := String" } EQ_Contact(in1 := #Serial_Number, in2 := #Functional_Tests_Panels[12].Serial_Number)
   END_RUNG wire#w2
   RUNG wire#w1
      { S7_Templates := "SrcType := String" } EQ_Contact(in1 := #Serial_Number, in2 := #Functional_Tests_Panels[13].Serial_Number)
   END_RUNG wire#w2
   RUNG wire#w1
      { S7_Templates := "SrcType := String" } EQ_Contact(in1 := #Serial_Number, in2 := #Functional_Tests_Panels[14].Serial_Number)
   END_RUNG wire#w2
   RUNG wire#w1
      { S7_Templates := "SrcType := String" } EQ_Contact(in1 := #Serial_Number, in2 := #Functional_Tests_Panels[15].Serial_Number)
   END_RUNG wire#w2
   RUNG wire#w1
      { S7_Templates := "SrcType := String" } EQ_Contact(in1 := #Serial_Number, in2 := #Functional_Tests_Panels[16].Serial_Number)
   END_RUNG wire#w2
   RUNG wire#w1
      { S7_Templates := "SrcType := String" } EQ_Contact(in1 := #Serial_Number, in2 := #Functional_Tests_Panels[17].Serial_Number)
   END_RUNG wire#w2
   RUNG wire#w1
      { S7_Templates := "SrcType := String" } EQ_Contact(in1 := #Serial_Number, in2 := #Functional_Tests_Panels[18].Serial_Number)
   END_RUNG wire#w2
   RUNG wire#w1
      { S7_Templates := "SrcType := String" } EQ_Contact(in1 := #Serial_Number, in2 := #Functional_Tests_Panels[19].Serial_Number)
   END_RUNG wire#w2
   RUNG wire#w1
      { S7_Templates := "SrcType := String" } EQ_Contact(in1 := #Serial_Number, in2 := #Functional_Tests_Panels[20].Serial_Number)
   END_RUNG wire#w2
   RUNG wire#w1
      { S7_Templates := "SrcType := String" } EQ_Contact(in1 := #Serial_Number, in2 := #Functional_Tests_Panels[21].Serial_Number)
   END_RUNG wire#w2
   RUNG wire#w1
      { S7_Templates := "SrcType := String" } EQ_Contact(in1 := #Serial_Number, in2 := #Functional_Tests_Panels[22].Serial_Number)
   END_RUNG wire#w2
   RUNG wire#w1
      { S7_Templates := "SrcType := String" } EQ_Contact(in1 := #Serial_Number, in2 := #Functional_Tests_Panels[23].Serial_Number)
   END_RUNG wire#w2
   RUNG wire#w1
      { S7_Templates := "SrcType := String" } EQ_Contact(in1 := #Serial_Number, in2 := #Functional_Tests_Panels[24].Serial_Number)
   END_RUNG wire#w2
   RUNG wire#w1
      { S7_Templates := "SrcType := String" } EQ_Contact(in1 := #Serial_Number, in2 := #Functional_Tests_Panels[25].Serial_Number)
   END_RUNG wire#w2
   RUNG wire#w1
      { S7_Templates := "SrcType := String" } EQ_Contact(in1 := #Serial_Number, in2 := #Functional_Tests_Panels[26].Serial_Number)
   END_RUNG wire#w2
   RUNG wire#w1
      { S7_Templates := "SrcType := String" } EQ_Contact(in1 := #Serial_Number, in2 := #Functional_Tests_Panels[27].Serial_Number)
   END_RUNG wire#w2
   RUNG wire#w1
      { S7_Templates := "SrcType := String" } EQ_Contact(in1 := #Serial_Number, in2 := #Functional_Tests_Panels[28].Serial_Number)
   END_RUNG wire#w2
   RUNG wire#w1
      { S7_Templates := "SrcType := String" } EQ_Contact(in1 := #Serial_Number, in2 := #Functional_Tests_Panels[29].Serial_Number)
   END_RUNG wire#w2
   RUNG wire#w1
      { S7_Templates := "SrcType := String" } EQ_Contact(in1 := #Serial_Number, in2 := #Functional_Tests_Panels[30].Serial_Number)
   END_RUNG wire#w2
   // the same network as SCL:
   #Got_Married := (#Serial_Number <> '') AND ((#Serial_Number = #Functional_Tests_Panels[1].Serial_Number) OR (#Serial_Number = #Functional_Tests_Panels[2].Serial_Number) OR (#Serial_Number = #Functional_Tests_Panels[3].Serial_Number) OR (#Serial_Number = #Functional_Tests_Panels[4].Serial_Number) OR (#Serial_Number = #Functional_Tests_Panels[5].Serial_Number) OR (#Serial_Number = #Functional_Tests_Panels[6].Serial_Number) OR (#Serial_Number = #Functional_Tests_Panels[7].Serial_Number) OR (#Serial_Number = #Functional_Tests_Panels[8].Serial_Number) OR (#Serial_Number = #Functional_Tests_Panels[9].Serial_Number) OR (#Serial_Number = #Functional_Tests_Panels[10].Serial_Number) OR (#Serial_Number = #Functional_Tests_Panels[11].Serial_Number) OR (#Serial_Number = #Functional_Tests_Panels[12].Serial_Number) OR (#Serial_Number = #Functional_Tests_Panels[13].Serial_Number) OR (#Serial_Number = #Functional_Tests_Panels[14].Serial_Number) OR (#Serial_Number = #Functional_Tests_Panels[15].Serial_Number) OR (#Serial_Number = #Functional_Tests_Panels[16].Serial_Number) OR (#Serial_Number = #Functional_Tests_Panels[17].Serial_Number) OR (#Serial_Number = #Functional_Tests_Panels[18].Serial_Number) OR (#Serial_Number = #Functional_Tests_Panels[19].Serial_Number) OR (#Serial_Number = #Functional_Tests_Panels[20].Serial_Number) OR (#Serial_Number = #Functional_Tests_Panels[21].Serial_Number) OR (#Serial_Number = #Functional_Tests_Panels[22].Serial_Number) OR (#Serial_Number = #Functional_Tests_Panels[23].Serial_Number) OR (#Serial_Number = #Functional_Tests_Panels[24].Serial_Number) OR (#Serial_Number = #Functional_Tests_Panels[25].Serial_Number) OR (#Serial_Number = #Functional_Tests_Panels[26].Serial_Number) OR (#Serial_Number = #Functional_Tests_Panels[27].Serial_Number) OR (#Serial_Number = #Functional_Tests_Panels[28].Serial_Number) OR (#Serial_Number = #Functional_Tests_Panels[29].Serial_Number) OR (#Serial_Number = #Functional_Tests_Panels[30].Serial_Number));
END_REGION
END_FUNCTION_BLOCK
